// TIA Portal project "Diarator_V2" (V16)

(* hardware
DEVICE "S7-1200 station_1"  S7-1200 Station
   slot 0: "Rack_0"  S7-1200 Rack  Rack  V1.0
   slot 1: "PLC_1"  CPU 1214C DC/DC/Rly  6ES7 214-1HG40-0XB0  V4.4
   slot 2: "DI 16/DQ 16x24VDC_2"  SM 1223 DI8/DQ8 x relay  6ES7 223-1PH32-0XB0  V2.0
   slot 3: "AI 4x13BIT_1"  6ES7 231-4HD32-0XB0  V2.1
   slot 4: "AI 4x13BIT_2"  6ES7 231-4HD32-0XB0  V2.1
   slot 5: "AQ 4x14BIT_1"  6ES7 232-4HD32-0XB0  V2.1
*)

// ===== PLC "PLC_1"  CPU 1214C DC/DC/Rly =====

VAR_GLOBAL   // PLC tag table "Default tag table"
   "rAlarm_SetMinPressSteam" AT %MW12 : Int;   // Уставка минимального давления пара
   "rAI_Press1" AT %MW14 : Int;   // Давление датчика
   "bAlarmPress1" AT %M16.0 : Bool;
   "rAlarm_SetMinPressWater" AT %MW18 : Int;   // Уставка аварийного давления воды
   "rAI_Press2" AT %MW20 : Int;
   "1_MTrig" AT %M6.4 : Bool;
   "2_MTrig" AT %M6.5 : Bool;
   "3_MTrig" AT %M6.6 : Bool;
   "mTrig1" AT %M7.0 : Bool;
   "mTrig" AT %M1.4 : Bool;
END_VAR

VAR_GLOBAL   // PLC tag table "HMI_"
   "bHMI_button_Start" AT %M2.0 : Bool;   // Кнопка старт
   "bHMI_button_Stop" AT %M2.1 : Bool;   // Кнопка стоп
   "bHMI_button_Pause" AT %M2.2 : Bool;   // Кнопка пауза
   "bStartAllowed" AT %M100.0 : Bool;   // Готовность к старту
   "bOpenWindStartConveyor" AT %M100.1 : Bool;   // Вызов окна подтверждения оператором старта конвейера
   "iHMI_Num_StatrPaster" AT %MW4 : Int;
   "bTypePID_Zone1" AT %M8.0 : Bool;   // Тип ПИД - 1 - Охлаждение, 0 - Нагрев
   "bTypePID_Zone2" AT %M8.1 : Bool;   // Тип ПИД - 1 - Охлаждение, 0 - Нагрев
   "bTypePID_Zone3" AT %M8.2 : Bool;   // Тип ПИД - 1 - Охлаждение, 0 - Нагрев
   "bTypePID_Zone4" AT %M8.3 : Bool;   // Тип ПИД - 1 - Охлаждение, 0 - Нагрев
   "bTypePID_Zone5" AT %M8.4 : Bool;   // Тип ПИД - 1 - Охлаждение, 0 - Нагрев
   "bAllAuto" AT %M0.6 : Bool;   // Перевод всего оборудования в авто с ручного
   "bZoomerOff" AT %M0.7 : Bool;   // Выкл пищалка
   "bResetAlarmCommon" AT %M6.0 : Bool;   // Общий сброс аварий
   "bResCountWaterO2" AT %M0.5 : Bool;   // Сброс счетчика готовой воды
   "bCountWaterToSewerge" AT %MW72 : Int;   // Счетчики воды в канализацию
   "bCountWaterToReadyO2" AT %MD10 : DInt;   // Счетчикиготовой водыО2
   "bHMI_ResetCounterAll_Water" AT %M3.2 : Bool;   // Кнопка сброса счетчика воды общего
   "iCount_All_Water" AT %MD62 : UDInt;   // Значение общего кол-ва воды пройденного через счетчик
   "iCount_CIP_AlL" AT %MD126 : UDInt;   // Счетчик СИП
   "bResCount_CIP" AT %M3.3 : Bool;   // Кнопка Сброса счетчика СИП
   "iStatusWork" AT %MW76 : Int;   // 0 - стоп 1 - СИП 2 - ДИаратор Подготовка 4 - Диаратор производство Статус работы для панели
   "timeStart" AT %MD50 : DInt;   // Задержка стоп/старт насосы
   "timeAlarmNoWater" AT %MD54 : DInt;   // Авария при длительной отстутвии воды
   "bDryContrlPump_1" AT %M78.0 : Bool;   // Контроль сухого хода насоса 1
   "bResTimeWorkSystem" AT %M6.7 : Bool;   // Сброс времени наработки системой
   "iOurs_WorkSystem" AT %MW120 : UInt;   // Часы работы системы
   "iMini_WorkSystem" AT %MW122 : Int;   // Мин работы системы
   "iSec_WorkSystem" AT %MW124 : Int;   // Секунды работы системы
END_VAR

VAR_GLOBAL   // PLC tag table "DI"
   "DI_0.0_Кнопка экстренной остановки E-Stop №1" AT %I0.0 : Bool;
   "DI_0.1_Положение ВОДА" AT %I0.1 : Bool;
   "DI_0.2_Положение СИП" AT %I0.2 : Bool;
   "DI_0.3_Клапан V1" AT %I0.3 : Bool;
   "DI_0.4_Клапан V3" AT %I0.4 : Bool;   // Импльс от расходомера
   "DI_0.5_Клапан V4" AT %I0.5 : Bool;
   "DI_0.6_Клапан V5" AT %I0.6 : Bool;
   "DI_0.7_Клапан V6" AT %I0.7 : Bool;
   "DI_1.0_LS1" AT %I1.0 : Bool;
   "DI_1.1_LS2" AT %I1.1 : Bool;
   "DI_1.2_LS3" AT %I1.2 : Bool;
   "DI_1.3_LS4" AT %I1.3 : Bool;
   "DI_1.4_Реле давления воздуха" AT %I1.4 : Bool;
   "DI_1.5_Импульсы Расходомера" AT %I1.5 : Bool;
   "DI_2.0_Автомат_1" AT %I2.0 : Bool;
   "DI_2.1_Работа_Частотник_1" AT %I2.1 : Bool;
   "DI_2.2_Автомат_2" AT %I2.2 : Bool;
   "DI_2.3_Работа_Частотник_2" AT %I2.3 : Bool;
END_VAR

VAR_GLOBAL   // PLC tag table "MyTags"
   "Разрешение работы конвейера" AT %M0.0 : Bool;   // Команда разрешения от Глобального блока работы
   "bMain_AlarmSystem" AT %M2.3 : Bool;   // АВария в системе (Общая)
   "bStartWork_Main" AT %M1.7 : Bool;   // Старт Общий Диаэратор
   "bPosition_Diarator" AT %M3.0 : Bool;   // Калачи в положении Диаэратор
   "bPosition_CIP" AT %M3.1 : Bool;   // Калачи в положении СИП
   "bReady_O2" AT %M1.3 : Bool;   // Готовность воды по датчику кислорода
   "bDiarator_WaterReady" AT %M0.2 : Bool;   // Меркер готовности диаратора по счетчику
   "bTypeControlO2" AT %M1.2 : Bool;   // Переключение типа контроля О2 (счетик - 0, датчик О2 - 1)
   "bImpulseFlow" AT %M3.4 : Bool;   // Импульс расходомера
   "diAccumTime" AT %MD116 : DInt;   // Аккумулятор времени работы установки
   "TestReset" AT %M7.1 : Bool;   // Блок аварий для тестов
   "bPaus" AT %M1.1 : Bool;
   "MTrig2" AT %M7.2 : Bool;
   "TestDI" AT %M0.4 : Bool;
   "m_STOP" AT %M1.6 : Bool;
   "_bCloseFV_CIP" AT %M1.0 : Bool;
END_VAR

VAR_GLOBAL   // PLC tag table "Timers_CPU"
   "Time_0.1s" AT %M500.0 : Bool;
   "Time_0.2s" AT %M500.1 : Bool;
   "Time_0.4s" AT %M500.2 : Bool;
   "Time_0.5s" AT %M500.3 : Bool;
   "Time_0.8s" AT %M500.4 : Bool;
   "Time_1s" AT %M500.5 : Bool;
   "Time_1.6s" AT %M500.6 : Bool;
   "Time_2s" AT %M500.7 : Bool;
END_VAR

VAR_GLOBAL   // PLC tag table "DO"
   "DO_0.0_Пневмо_остров клапан 1" AT %Q0.0 : Bool;
   "DO_0.1_Пневмо_остров клапан 2" AT %Q0.1 : Bool;
   "DO_0.2_Пневмо_остров клапан 3" AT %Q0.2 : Bool;
   "DO_0.3_Пневмо_остров клапан 4" AT %Q0.3 : Bool;
   "DO_0.4_Пневмо_остров клапан 5" AT %Q0.4 : Bool;
   "DO_0.5_Пневмо_остров клапан 6" AT %Q0.5 : Bool;
   "DO_0.6_Пневмо_остров клапан 7" AT %Q0.6 : Bool;
   "DO_0.7_Пневмо_остров клапан 8" AT %Q0.7 : Bool;
   "DO_0.8_Пневмо_остров клапан 9" AT %Q1.0 : Bool;
   "DO_0.9_Пневмо_остров клапан 10" AT %Q1.1 : Bool;
   "Преобразователь частоты 1 пуск" AT %Q2.4 : Bool;
   "Преобразователь частоты 2 пуск" AT %Q2.5 : Bool;
   "Световая колонна - зеленый" AT %Q2.0 : Bool;
   "Световая колонна - желтый" AT %Q2.1 : Bool;
   "Световая колонна - красный" AT %Q2.2 : Bool;
   "Выход_Готовность ВОДА" AT %Q2.6 : Bool;
   "Выход_Готовность СИП" AT %Q2.7 : Bool;
END_VAR

VAR_GLOBAL   // PLC tag table "AI"
   "ТТ01" AT %IW120 : Int;   // Температура
   "FIC" AT %IW112 : Int;   // Расходомер
   "PT-01" AT %IW114 : Int;   // Давление 1
   "PT-02" AT %IW116 : Int;   // Давление 2
   "PT-03" AT %IW118 : Int;   // Давление 3
   "O2" AT %IW124 : Int;   // Датчик Кислорода О2
   "ТТ02_FromO2" AT %IW126 : Int;   // Температура
END_VAR

VAR_GLOBAL   // PLC tag table "AO"
   "AO_0.0_Преобразователь частоты 1" AT %QW144 : Int;
   "AO_0.1_Преобразователь частоты 2" AT %QW146 : Int;
   "AO_0.2_Управляемый клапан №2" AT %QW148 : Int;
END_VAR

VAR_GLOBAL   // PLC tag table "_TEst_1"
   "test_stateDiar" AT %M0.1 : Bool;
   "test_PressSensor" AT %MD22 : Real;
END_VAR

TYPE "FV_o/c"
   STRUCT
      bOpenCmd : Bool;   // Команда открыть (автомат)
      bManualMode : Bool;   // Ручной режим (TRUE)
      bManualOpen : Bool;   // Команда открыть в ручном режиме
      bFeedbackOpen : Bool;   // Обратная связь "Открыт"
      tMaxTime : DInt;   // Время на открытие
      bResetAlarm : Bool;   // Сброс аварии
      bCheckFeedback : Bool;   // Выбирается есть ли обратная связь у клапана
      bOutOpen : Bool;   // Выход на открытие клапана
      iOutState : Int;   // Выход статуса клапана
   END_STRUCT;
END_TYPE

TYPE "PID_Param"
   STRUCT
      bModeActivate : Bool;   // Запуск выбранного типа работы
      iModeNum : Int := 3;   // 0 -стоп 1 - автонастройка 2 -точная автонастройка 3 - авто режим 4 - ручной режим
      iOutState : Int;   // В каком режиме ПИД
      bOutError : Bool;   // Выход при ошибке TRUE
      iOutErrorBits : Int;   // Бит с кодом ошибки (см. мануал)
      iProgress : Int;   // Состояние в % при автонастройки, сколько сделано
   END_STRUCT;
END_TYPE

TYPE "FV_regul"
   STRUCT
      bHMI_ManualMode : Bool;   // Переключение режима авто/ручно (0 - А, 1 - Р)
      rHMI_ManualSet : Real;   // Уставка в ручном режиме (0-100)
      rAuto_Set : Real;   // Уставка в автоматическом режиме
      iOut_AO : Int;   // Сигнал на аналоговый выход
      "rHMI_Out_FV-%" : Real;   // Состояние в % (0-100)
      bOut_DO_ValveOpen : Bool;   // Дискретный сигнал открытия
   END_STRUCT;
END_TYPE

TYPE "Коэф ПИД"
   STRUCT
      Gain : Int;   // Коэф П
      I : DInt;   // Коэф И
      D : DInt;   // Коэф Д
   END_STRUCT;
END_TYPE

TYPE "tipe_Pumps"
   STRUCT
      bAutoStartPump : Bool;   // Старт в автоматическом режиме
      rAutoSpeedPump : Real;   // Скорость в автоматическом режиме
      bManualMode : Bool;   // Ручной режим вкл/выкл
      bManualStart : Bool;   // Старт в ручном режиме
      rManualSpeed : Real;   // Скорость в ручном режиме
      rHMI_Speed : Real;   // Выходная скороость для HMI
      bHMI_PumpRun : Bool;   // Статус работы для HMI
      bresAlarm : Bool;   // Сброс аварий
      iStatusPump : Int;   // Статус насоса
   END_STRUCT;
END_TYPE

TYPE "Tipe_DI"
   STRUCT
      f_DI_out : Bool;
      "bFiltr_on/off" : Bool := true;
      diTime_filtr : Time := T#100ms;
      bSimulation : Bool;   // Включение режима симуляции
      "bSim_On/Off" : Bool;   // Управление симуляцией
   END_STRUCT;
END_TYPE

TYPE "Tipe_AI"
   STRUCT
      bSimulate : Bool;   // Вкл симуляции датчика
      rSimulateValue : Real;   // Значение симуляции датчика
      rSensor_HL : Real;   // Верхний предел датчика
      rSensor_LL : Real;   // Нижний предел датчика
      bFiltr : Bool;   // Управление фильтром значений
      rAI_Value : Real;   // Значение аналогового датчика
   END_STRUCT;
END_TYPE

// folder: AI_Signal/AI_DB/4-20

DATA_BLOCK "AI_(4-20)_1_DB_1"   // DB16
{ S7_Optimized_Access := 'FALSE' }
VERSION : 0.1
// stored: InstanceOfName AI_(4-20)_1
"AI_(4-20)_1"
BEGIN
   HMI_rParam_Sensor_HL := 100.0;
   HMI_rParam_Sensor_LL := -50.0;
END_DATA_BLOCK

DATA_BLOCK "AI_(4-20)_1_DB_2"   // DB17
{ S7_Optimized_Access := 'FALSE' }
VERSION : 0.1
// stored: InstanceOfName AI_(4-20)_1
"AI_(4-20)_1"
BEGIN
END_DATA_BLOCK

DATA_BLOCK "AI_(4-20)_1_DB_4"   // DB18
{ S7_Optimized_Access := 'FALSE' }
VERSION : 0.1
// stored: InstanceOfName AI_(4-20)_1
"AI_(4-20)_1"
BEGIN
   HMI_rParam_Sensor_HL := 6.0;
END_DATA_BLOCK

DATA_BLOCK "AI_(4-20)_1_DB_3"   // DB27
{ S7_Optimized_Access := 'FALSE' }
VERSION : 0.1
// stored: InstanceOfName AI_(4-20)_1
"AI_(4-20)_1"
BEGIN
   HMI_rParam_Sensor_HL := 100.0;
END_DATA_BLOCK

DATA_BLOCK "AI_(4-20)_1_DB_5"   // DB28
{ S7_Optimized_Access := 'FALSE' }
VERSION : 0.1
// stored: InstanceOfName AI_(4-20)_1
"AI_(4-20)_1"
BEGIN
   HMI_rParam_Sensor_HL := 6.0;
END_DATA_BLOCK

DATA_BLOCK "AI_(4-20)_1_DB_6"   // DB60
{ S7_Optimized_Access := 'FALSE' }
VERSION : 0.1
// stored: InstanceOfName AI_(4-20)_1
"AI_(4-20)_1"
BEGIN
END_DATA_BLOCK

DATA_BLOCK "AI_(4-20)_1_DB_7"   // DB61
{ S7_Optimized_Access := 'FALSE' }
VERSION : 0.1
// stored: InstanceOfName AI_(4-20)_1
"AI_(4-20)_1"
BEGIN
END_DATA_BLOCK

// folder: DB-FB

DATA_BLOCK "FB_check_For_Start_DB"   // DB1
{ S7_Optimized_Access := 'FALSE' }
VERSION : 0.1
// stored: InstanceOfName FB_check_For_Start
"FB_check_For_Start"
BEGIN
END_DATA_BLOCK

DATA_BLOCK "FB_Emergency_DB"   // DB3
{ S7_Optimized_Access := 'FALSE' }
VERSION : 0.1
// stored: InstanceOfName FB_Аварии
"FB_Аварии"
BEGIN
END_DATA_BLOCK

DATA_BLOCK "Tank_Diarator_DB"   // DB11
{ S7_Optimized_Access := 'TRUE' }
VERSION : 0.1
// stored: InstanceOfName Tank_Diarator
"Tank_Diarator"
BEGIN
END_DATA_BLOCK

DATA_BLOCK "FB_Control_O2_DB"   // DB12
{ S7_Optimized_Access := 'TRUE' }
VERSION : 0.1
// stored: InstanceOfName FB_Control_O2
"FB_Control_O2"
BEGIN
END_DATA_BLOCK

DATA_BLOCK "FB_Tank_2(Buffer)_DB"   // DB13
{ S7_Optimized_Access := 'TRUE' }
VERSION : 0.1
// stored: InstanceOfName FB_Tank_2(Buffer)
"FB_Tank_2(Buffer)"
BEGIN
END_DATA_BLOCK

DATA_BLOCK "FB_Control_Press_Tank2_DB"   // DB14
{ S7_Optimized_Access := 'TRUE' }
VERSION : 0.1
// stored: InstanceOfName FB_Control_Press_Tank2
"FB_Control_Press_Tank2"
BEGIN
END_DATA_BLOCK

DATA_BLOCK "FB_CIP_DB"   // DB15
{ S7_Optimized_Access := 'TRUE' }
VERSION : 0.1
// stored: InstanceOfName FB_CIP
"FB_CIP"
BEGIN
END_DATA_BLOCK

DATA_BLOCK "FB_OwerPress_Tank_2_DB"   // DB64
{ S7_Optimized_Access := 'FALSE' }
VERSION : 0.1
// stored: InstanceOfName FB_OwerPress_Tank_2
"FB_OwerPress_Tank_2"
BEGIN
END_DATA_BLOCK

DATA_BLOCK "FB_SVETOFOR_DB"   // DB102
{ S7_Optimized_Access := 'TRUE' }
VERSION : 0.1
// stored: InstanceOfName FB_SVETOFOR
"FB_SVETOFOR"
BEGIN
END_DATA_BLOCK

// folder: DI_signal/DB_DI

DATA_BLOCK "LS-1"   // DB33
{ S7_Optimized_Access := 'FALSE' }
VERSION : 0.1
// stored: InstanceOfName FB_DI_Pointer
"FB_DI_Pointer"
BEGIN
END_DATA_BLOCK

DATA_BLOCK "LS-2"   // DB35
{ S7_Optimized_Access := 'FALSE' }
VERSION : 0.1
// stored: InstanceOfName FB_DI_Pointer
"FB_DI_Pointer"
BEGIN
END_DATA_BLOCK

DATA_BLOCK "LS-3"   // DB36
{ S7_Optimized_Access := 'FALSE' }
VERSION : 0.1
// stored: InstanceOfName FB_DI_Pointer
"FB_DI_Pointer"
BEGIN
END_DATA_BLOCK

DATA_BLOCK "LS-4"   // DB46
{ S7_Optimized_Access := 'FALSE' }
VERSION : 0.1
// stored: InstanceOfName FB_DI_Pointer
"FB_DI_Pointer"
BEGIN
END_DATA_BLOCK

DATA_BLOCK "P1_ControlWorking"   // DB47
{ S7_Optimized_Access := 'FALSE' }
VERSION : 0.1
// stored: InstanceOfName FB_DI_Pointer
"FB_DI_Pointer"
BEGIN
END_DATA_BLOCK

DATA_BLOCK "DI_EStop1"   // DB48
{ S7_Optimized_Access := 'FALSE' }
VERSION : 0.1
// stored: InstanceOfName FB_DI
"FB_DI"
BEGIN
END_DATA_BLOCK

DATA_BLOCK "State_Water"   // DB49
{ S7_Optimized_Access := 'FALSE' }
VERSION : 0.1
// stored: InstanceOfName FB_DI
"FB_DI"
BEGIN
END_DATA_BLOCK

DATA_BLOCK "State_CIP"   // DB50
{ S7_Optimized_Access := 'FALSE' }
VERSION : 0.1
// stored: InstanceOfName FB_DI
"FB_DI"
BEGIN
END_DATA_BLOCK

DATA_BLOCK "FeedBack_V1"   // DB51
{ S7_Optimized_Access := 'FALSE' }
VERSION : 0.1
// stored: InstanceOfName FB_DI
"FB_DI"
BEGIN
END_DATA_BLOCK

DATA_BLOCK "Feedback_V3"   // DB52
{ S7_Optimized_Access := 'FALSE' }
VERSION : 0.1
// stored: InstanceOfName FB_DI
"FB_DI"
BEGIN
END_DATA_BLOCK

DATA_BLOCK "Feedback_V4"   // DB53
{ S7_Optimized_Access := 'FALSE' }
VERSION : 0.1
// stored: InstanceOfName FB_DI
"FB_DI"
BEGIN
END_DATA_BLOCK

DATA_BLOCK "FeedBack_V5"   // DB54
{ S7_Optimized_Access := 'FALSE' }
VERSION : 0.1
// stored: InstanceOfName FB_DI
"FB_DI"
BEGIN
END_DATA_BLOCK

DATA_BLOCK "FeedBack_V6"   // DB55
{ S7_Optimized_Access := 'FALSE' }
VERSION : 0.1
// stored: InstanceOfName FB_DI
"FB_DI"
BEGIN
END_DATA_BLOCK

DATA_BLOCK "PressAir"   // DB78
{ S7_Optimized_Access := 'FALSE' }
VERSION : 0.1
// stored: InstanceOfName FB_DI_Pointer
"FB_DI_Pointer"
BEGIN
END_DATA_BLOCK

DATA_BLOCK "ImpFlow"   // DB79
{ S7_Optimized_Access := 'FALSE' }
VERSION : 0.1
// stored: InstanceOfName FB_DI_Pointer
"FB_DI_Pointer"
BEGIN
END_DATA_BLOCK

DATA_BLOCK "CircuitControl-1"   // DB80
{ S7_Optimized_Access := 'FALSE' }
VERSION : 0.1
// stored: InstanceOfName FB_DI_Pointer
"FB_DI_Pointer"
BEGIN
END_DATA_BLOCK

DATA_BLOCK "CircuitControl-2"   // DB81
{ S7_Optimized_Access := 'FALSE' }
VERSION : 0.1
// stored: InstanceOfName FB_DI_Pointer
"FB_DI_Pointer"
BEGIN
END_DATA_BLOCK

DATA_BLOCK "P2_ControlWorking"   // DB82
{ S7_Optimized_Access := 'FALSE' }
VERSION : 0.1
// stored: InstanceOfName FB_DI_Pointer
"FB_DI_Pointer"
BEGIN
END_DATA_BLOCK

// folder: FB/R_TRIG_DB

DATA_BLOCK "R_trig_All_Auto"   // DB40
{ S7_Optimized_Access := 'TRUE' }
VERSION : 0.1
// stored: InstanceOfName R_trig
"R_trig"
BEGIN
END_DATA_BLOCK

DATA_BLOCK "R_trig_DB_Stop_CIP"   // DB56
{ S7_Optimized_Access := 'TRUE' }
VERSION : 0.1
// stored: InstanceOfName R_trig
"R_trig"
BEGIN
END_DATA_BLOCK

DATA_BLOCK "R_trig_ResTimeWorkSystem"   // DB58
{ S7_Optimized_Access := 'TRUE' }
VERSION : 0.1
// stored: InstanceOfName R_trig
"R_trig"
BEGIN
END_DATA_BLOCK

DATA_BLOCK "R_trig_DB"   // DB99
{ S7_Optimized_Access := 'TRUE' }
VERSION : 0.1
// stored: InstanceOfName R_trig
"R_trig"
BEGIN
END_DATA_BLOCK

DATA_BLOCK "R_trig_DB_Alarm_Zoomer"   // DB101
{ S7_Optimized_Access := 'TRUE' }
VERSION : 0.1
// stored: InstanceOfName R_trig
"R_trig"
BEGIN
END_DATA_BLOCK

DATA_BLOCK "R_trig_DB_Pause"   // DB103
{ S7_Optimized_Access := 'TRUE' }
VERSION : 0.1
// stored: InstanceOfName R_trig
"R_trig"
BEGIN
END_DATA_BLOCK

// folder: System blocks/Program resources

DATA_BLOCK "IEC_Counter_ReadyWaterO2"   // DB29
{ S7_Optimized_Access := 'TRUE' }
AUTHOR : SIMATIC
FAMILY : IEC
NAME : DCNTR
VERSION : 1.2
// stored: InstanceOfName IEC_DCOUNTER
"IEC_DCOUNTER"
BEGIN
END_DATA_BLOCK

DATA_BLOCK "IEC_Counter_DiarSewerage"   // DB31
{ S7_Optimized_Access := 'TRUE' }
AUTHOR : Simatic
FAMILY : IEC
NAME : CNTR
VERSION : 1.0
// stored: InstanceOfName IEC_COUNTER
"IEC_COUNTER"
BEGIN
END_DATA_BLOCK

DATA_BLOCK "IEC_Counter_All_Water"   // DB37
{ S7_Optimized_Access := 'TRUE' }
AUTHOR : Simatic
FAMILY : IEC
NAME : UDCNTR
VERSION : 1.2
// stored: InstanceOfName IEC_UDCOUNTER
"IEC_UDCOUNTER"
BEGIN
END_DATA_BLOCK

DATA_BLOCK "IEC_Counter_CIP"   // DB38
{ S7_Optimized_Access := 'TRUE' }
AUTHOR : Simatic
FAMILY : IEC
NAME : UCNTR
VERSION : 1.2
// stored: InstanceOfName IEC_UCOUNTER
"IEC_UCOUNTER"
BEGIN
END_DATA_BLOCK

DATA_BLOCK "IEC_Timer_DetectDry_1"   // DB42
{ S7_Optimized_Access := 'TRUE' }
AUTHOR : Simatic
FAMILY : IEC
NAME : IEC_TMR
VERSION : 1.0
// stored: InstanceOfName IEC_TIMER
"IEC_TIMER"
BEGIN
END_DATA_BLOCK

DATA_BLOCK "IEC_Timer_ResDrySens"   // DB45
{ S7_Optimized_Access := 'TRUE' }
AUTHOR : Simatic
FAMILY : IEC
NAME : IEC_TMR
VERSION : 1.0
// stored: InstanceOfName IEC_TIMER
"IEC_TIMER"
BEGIN
END_DATA_BLOCK

DATA_BLOCK "IEC_Counter_0_DB"   // DB59
{ S7_Optimized_Access := 'TRUE' }
AUTHOR : Simatic
FAMILY : IEC
NAME : CNTR
VERSION : 1.0
// stored: InstanceOfName IEC_COUNTER
"IEC_COUNTER"
BEGIN
END_DATA_BLOCK

DATA_BLOCK "IEC_Timer_0_DB"   // DB62
{ S7_Optimized_Access := 'TRUE' }
AUTHOR : Simatic
FAMILY : IEC
NAME : IEC_TMR
VERSION : 1.0
// stored: InstanceOfName IEC_TIMER
"IEC_TIMER"
BEGIN
END_DATA_BLOCK

// folder: Use VARs to HMI

DATA_BLOCK "DB2_HMI_SET"   // DB2
{ S7_Optimized_Access := 'FALSE' }
VERSION : 0.1
   VAR
      rO2_SP : Real;   // Уставка для датчика кислорода
      rHisteresis_O2_SP : Real;   // Уставка гистерезиса для допустим отклонения О2
      diTimeLost_Gist_O2 : DInt;   // Уставка времени ожидания при выходе за пределы уставки
      rFlow_SP : Int;   // Уставка расхода воды готовности по счетчику
      diTimeToReadyO2 : DInt;   // Уставка ожидания перехода в готовность воды при достижении уставки О2
      rPT02_SP : Real;   // Уставка давления в танке 2
      rPT02_OwerPress_SP : Real;   // Уставка слишком высокого давления Танк 2
      rPT02_Hister_OwerPress : Real;   // Уставка гистерезиса
      diTimeToOpenValveCO2 : DInt := 2;   // Время отсчета для открытия клапана при понижении давления в Такнке 2
      diTimeToCloseValveCO2 : DInt := 2;   // Время отсчета для закрытия клапана при возвращении давления в Такнке 2
      diFlipTimeCIP : DInt := 3;   // Время задержки между переходом флипования
      diFlipPauseFlipeCIP : DInt := 2;   // Время задержки перед началом цикла флипования
      rSetValve_2_OUT : Real;   // Уставка расхода для клапана 2 задание для клапана
      rSetValve_2_Diarator : Real := 3000.0;   // Уставка клапана 2 при режиме ДИаратор
      rSetValve_2_CIP : Real := 5000.0;   // Уставка клапана 2 при режиме СИП
      "rSetPump-1_OUT" : Real;   // Уставка для насоса 1 - OUT
      "rSetPump-1_Diarator" : Real := 30.0;   // Уставка для насоса 1 - Диаратор
      "rSetPump-1_CIP" : Real := 20.0;   // Уставка для насоса 1 - CIP
      "rSetPump-2_OUT" : Real;   // Уставка для насоса 2 - OUT
      "rSetPump-2_Diarator" : Real := 3.0;   // Уставка для насоса 2 - Диаратор
      "rSetPump-2_CIP" : Real := 3.0;   // Уставка для насоса 2 - CIP
      rDetectDry_PressTank1_SP : Real := 2.0;   // Уставка обнаружения сухого хода для насоса 1
      diTimeDetectDrt : DInt := 2;   // Время для обнаружения сухого хода
      Di_timeCloseFV : DInt := 5000;   // Время задержки закрытия клапанов в режиме СИП при "СТОП"
      rLewelTank1_Stop : Real;   // Уровень емкости - закрытие Кл1
      rLewelTank1_Start : Real;   // Уровень емкости - открытие Кл1
   END_VAR
BEGIN
END_DATA_BLOCK

DATA_BLOCK "FVs_o/p"   // DB6
{ S7_Optimized_Access := 'FALSE' }
VERSION : 0.1
   VAR
      FV_1 : "FV_o/c";
      FV_2 : "FV_o/c";
      FV_3 : "FV_o/c";
      FV_4 : "FV_o/c";
      FV_5 : "FV_o/c";
      FV_6 : "FV_o/c";
      FV_7 : "FV_o/c";
      FV_8 : "FV_o/c";
      FV_9 : "FV_o/c";
      FV_10 : "FV_o/c";
   END_VAR
BEGIN
END_DATA_BLOCK

DATA_BLOCK "FVs_Regul"   // DB24
{ S7_Optimized_Access := 'FALSE' }
VERSION : 0.1
   VAR
      FV_Regul_1 : "FV_regul";
   END_VAR
BEGIN
END_DATA_BLOCK

DATA_BLOCK "Pumps"   // DB30
{ S7_Optimized_Access := 'FALSE' }
VERSION : 0.1
   VAR
      Pump_1 : "tipe_Pumps";
      Pump_2 : "tipe_Pumps";
   END_VAR
BEGIN
END_DATA_BLOCK

DATA_BLOCK "LS"   // DB34
{ S7_Optimized_Access := 'FALSE' }
VERSION : 0.1
   VAR
      "LS-1" : Bool;   // Уровень емкости 1 колонны
      "LS-2" : Bool;   // Нижний уровень 2 колонны
      "LS-3" : Bool;   // Средний уровень 2 колонны
      "LS-4" : Bool;   // Верхний уровень 2 колонны
   END_VAR
BEGIN
END_DATA_BLOCK

DATA_BLOCK "DI"   // DB43
{ S7_Optimized_Access := 'FALSE' }
VERSION : 0.1
   VAR
      DI_0 : "Tipe_DI";   // Stop_Button
      DI_1 : "Tipe_DI";   // Water_State
      DI_2 : "Tipe_DI";   // CIP_State
      DI_3 : "Tipe_DI";   // Feedback_V1
      DI_4 : "Tipe_DI";   // Feedback_V3
      DI_5 : "Tipe_DI";   // Feedback_V4
      DI_6 : "Tipe_DI";   // Feedback_V5
      DI_7 : "Tipe_DI";   // Feedback_V6
      DI_8 : "Tipe_DI";   // LS-1
      DI_9 : "Tipe_DI";   // LS-2
      DI_10 : "Tipe_DI";   // LS-3
      DI_11 : "Tipe_DI";   // LS-4
      DI_12 : "Tipe_DI";   // PressAir_Rele
      DI_13 : "Tipe_DI";   // Impuls_CounterFlow
      DI_14 : "Tipe_DI";   // Доп контакт автомата 1
      DI_15 : "Tipe_DI";   // StatusWorkPump1
      DI_16 : "Tipe_DI";   // Доп контакт автомата 2
      DI_17 : "Tipe_DI";   // StatusWorkPump2
      DI_18 : "Tipe_DI";
      DI_19 : "Tipe_DI";
      DI_20 : "Tipe_DI";
      DI_21 : "Tipe_DI";
      DI_22 : "Tipe_DI";
      DI_23 : "Tipe_DI";
      DI_24 : "Tipe_DI";
      DI_25 : "Tipe_DI";
      DI_26 : "Tipe_DI";
      DI_27 : "Tipe_DI";
      DI_28 : "Tipe_DI";
      DI_29 : "Tipe_DI";
      DI_30 : "Tipe_DI";
   END_VAR
BEGIN
END_DATA_BLOCK

DATA_BLOCK "PID_State_Param"   // DB57
{ S7_Optimized_Access := 'FALSE' }
VERSION : 0.1
   VAR
      PID_Vavle2 : "PID_Param";
      PID_Pump1 : "PID_Param";
      PID_Pump2 : "PID_Param";
   END_VAR
BEGIN
END_DATA_BLOCK

DATA_BLOCK "Alarms"   // DB87
{ S7_Optimized_Access := 'FALSE' }
VERSION : 0.1
   VAR
      Ai_Alarm : Array[1..8] of Struct   // Аварии датчиков аналоговых
         ALARM : Bool;
         RESET : Bool;
      END_STRUCT;
      Pump_Alarm : Array[1..5] of Struct   // Аварии насосов
         ALARM : Bool;
         RESET : Bool;
      END_STRUCT;
      Avtomat_Off : Array[1..2] of Struct   // Контроль состояния вкл мотор автоматов
         ALARM : Bool;
      END_STRUCT;
      FV_Alarm : Array[1..10] of Struct   // Авария клапанов
         ALARM : Bool;
         RESET : Bool;
      END_STRUCT;
      "xE-Stop_1" : Bool;   // Авария по кнопке 1
      xVoltRele : Bool;   // Авария реле контроля фаз
      xLongWaitWater : Bool;   // Авария, долгое ожидание заполнения нижнего уровня емкости
      xPressAir : Bool;   // Авария реле давления воздуха
   END_VAR
BEGIN
END_DATA_BLOCK

DATA_BLOCK "AI_DB"   // DB90
{ S7_Optimized_Access := 'FALSE' }
VERSION : 0.1
   VAR
      TT_01 : "Tipe_AI";   // Температура
      FIC : "Tipe_AI";   // Расходомер
      PT_01 : "Tipe_AI";   // Давление Емкость_1
      PT_02 : "Tipe_AI";   // Давление Емкость_2
      PT_03 : "Tipe_AI";   // Давление Выход с емкости
      ТТ02_FromO2 : "Tipe_AI";   // Значение температуры с датчика кислорода
      O2 : "Tipe_AI";   // Кислород
   END_VAR
BEGIN
   O2.rSensor_HL := 10.0;
   O2.bFiltr := true;
   TT_01.bFiltr := true;
   FIC.bFiltr := true;
   PT_01.bFiltr := true;
   PT_02.bFiltr := true;
   PT_03.bFiltr := true;
   TT_01.rSensor_HL := 100.0;
   TT_01.rSensor_LL := -50.0;
   PT_01.rSensor_HL := 1.0;
   PT_02.rSensor_HL := 6.0;
   PT_03.rSensor_HL := 6.0;
END_DATA_BLOCK

// folder: Клапана/FV_o/C/FV_DB

DATA_BLOCK "FV_1"   // DB4
{ S7_Optimized_Access := 'FALSE' }
VERSION : 0.1
// stored: InstanceOfName Valve(c/o)
"Valve(c/o)"
BEGIN
END_DATA_BLOCK

DATA_BLOCK "FV_5"   // DB5
{ S7_Optimized_Access := 'FALSE' }
VERSION : 0.1
// stored: InstanceOfName Valve(c/o)
"Valve(c/o)"
BEGIN
END_DATA_BLOCK

DATA_BLOCK "FV_6"   // DB7
{ S7_Optimized_Access := 'FALSE' }
VERSION : 0.1
// stored: InstanceOfName Valve(c/o)
"Valve(c/o)"
BEGIN
END_DATA_BLOCK

DATA_BLOCK "FV_7"   // DB8
{ S7_Optimized_Access := 'FALSE' }
VERSION : 0.1
// stored: InstanceOfName Valve(c/o)
"Valve(c/o)"
BEGIN
END_DATA_BLOCK

DATA_BLOCK "FV_2"   // DB9
{ S7_Optimized_Access := 'FALSE' }
VERSION : 0.1
// stored: InstanceOfName Valve(c/o)
"Valve(c/o)"
BEGIN
END_DATA_BLOCK

DATA_BLOCK "FV_3"   // DB10
{ S7_Optimized_Access := 'FALSE' }
VERSION : 0.1
// stored: InstanceOfName Valve(c/o)
"Valve(c/o)"
BEGIN
END_DATA_BLOCK

DATA_BLOCK "FV_4"   // DB19
{ S7_Optimized_Access := 'FALSE' }
VERSION : 0.1
// stored: InstanceOfName Valve(c/o)
"Valve(c/o)"
BEGIN
END_DATA_BLOCK

DATA_BLOCK "FV_8"   // DB21
{ S7_Optimized_Access := 'FALSE' }
VERSION : 0.1
// stored: InstanceOfName Valve(c/o)
"Valve(c/o)"
BEGIN
END_DATA_BLOCK

DATA_BLOCK "FV_9"   // DB22
{ S7_Optimized_Access := 'FALSE' }
VERSION : 0.1
// stored: InstanceOfName Valve(c/o)
"Valve(c/o)"
BEGIN
END_DATA_BLOCK

DATA_BLOCK "FV_10"   // DB23
{ S7_Optimized_Access := 'FALSE' }
VERSION : 0.1
// stored: InstanceOfName Valve(c/o)
"Valve(c/o)"
BEGIN
END_DATA_BLOCK

// folder: Клапана/FV_regul/DB

DATA_BLOCK "FV_Regul_1_DB"   // DB20
{ S7_Optimized_Access := 'FALSE' }
VERSION : 0.1
// stored: InstanceOfName Valve(regul)
"Valve(regul)"
BEGIN
END_DATA_BLOCK

// folder: Насосы/DB

DATA_BLOCK "Pump_1_DB"   // DB25
{ S7_Optimized_Access := 'FALSE' }
VERSION : 0.1
// stored: InstanceOfName Pump
"Pump"
BEGIN
END_DATA_BLOCK

DATA_BLOCK "Pump_2_DB"   // DB26
{ S7_Optimized_Access := 'FALSE' }
VERSION : 0.1
// stored: InstanceOfName Pump
"Pump"
BEGIN
END_DATA_BLOCK

// folder: (top level)

FUNCTION_BLOCK "Tank_Diarator"   // FB2, SCL
{ S7_Optimized_Access := 'TRUE' }
VERSION : 0.1
   VAR_INPUT
      bEnable : Bool;   // Разрешение на работу
      bPause : Bool;   // Остановка производства воды
      bReady_O2 : Bool;   // Готовность воды по датчику О2
      bControlO2_Type : Bool;   // 1 = по СО2, 0 по расходу. Тип контроля кол-ва кислорода (датчик, или расход)
      rPT01 : Real;   // Значение давления РТ01
      iРасход_Накопленный : Int;   // Значение накопленного расхода воды
      iFlow_SP : Int := 10;   // Уставка для Расхода по счетчику
      diTimeWaitingReadyO2 : DInt := 30;   // Времы выдержки до маркера готовности по датчику О2
   END_VAR
   VAR_OUTPUT
      bValve1 : Bool;   // Клапан набор
      bValve2 : Bool;   // Клапан регуллирующий, разрешение на работу
      bValve3 : Bool;   // Клапан слива в дренаж
      bValve5 : Bool;   // Клапан набора готовой воды в емкость
      bValve7 : Bool;   // Клапан СО2 в емкость подготовки
      bWaterReady : Bool;   // Маркер готовности воды
      bPump_1 : Bool;   // Разрешение на работу насоса
   END_VAR
   VAR RETAIN
      TON_ready_O2 : TON_TIME;   // Таймер готовности по датчику кислорода
   END_VAR
BEGIN
   //Перевод из мс в Сек для таймера ожидания О2
   #diTimeWaitingReadyO2 := #diTimeWaitingReadyO2 * 1000;

   //Начало если нет разрешения на работу
   IF NOT #bEnable THEN
       //Закрываем все клапана
       #bValve1 := #bValve2 := #bValve3 := #bValve5 := #bValve7 := FALSE;
       // Стоп насоса
       #bPump_1 := FALSE;
       //Нет работы сброс всего
       #bWaterReady := FALSE;
       #TON_ready_O2.IN := FALSE;
       RETURN;
   END_IF;

   //Начало работы блока если есть разрешение

   //Подача клапан 1
   IF #rPT01 >= "DB2_HMI_SET".rLewelTank1_Stop THEN
       #bValve1 := FALSE;
   ELSIF #rPT01 <= "DB2_HMI_SET".rLewelTank1_Start THEN
       #bValve1 := TRUE;
   END_IF;

   //#bValve1 := TRUE;   
   #bValve2 := TRUE;   //Регулятор расхода для емкости (ПИД разрешение работы)
   #bValve3 := TRUE;   //Слив воды в дренаж, пока вода не будет подготовлена
   #bValve7 := TRUE;   //Co2
   #bPump_1 := TRUE;   //Разрешение на работу ПИД насоса по датчику давления в емкости

   //Проверка выбора типа контроля уровня кислорода

   IF #bControlO2_Type THEN
       #TON_ready_O2(IN:= #bReady_O2, PT := #diTimeWaitingReadyO2, Q =>#bWaterReady);   //Время выдержки при достижении уставки по О2
   ELSE
       #bWaterReady := (#iРасход_Накопленный >= #iFlow_SP);
   END_IF;

   IF #bWaterReady THEN
       #bValve3 := FALSE;  //Слив в дренаж
       #bValve5 := TRUE;   //Подача воды в емкость
   ELSE
       #bValve3 := TRUE;  //Слив в дренаж
       #bValve5 := FALSE;   //Подача воды в емкость
   END_IF;

   IF #bPause THEN
       #bValve1 := #bValve2 := #bValve3 := #bValve5 := #bValve7 := FALSE;
       #bPump_1 := FALSE;
       //Нет работы сброс всего
       #bWaterReady := FALSE;
       //Сброс таймера
       #TON_ready_O2.IN := FALSE;
   END_IF;
END_FUNCTION_BLOCK

FUNCTION_BLOCK "FB_Control_O2"   // FB6, SCL
{ S7_Optimized_Access := 'TRUE' }
VERSION : 0.1
   VAR_INPUT
      bEnable : Bool;
      rO2_SP : Real;   // Уставка О2
      rO2_Actual : Real;   // Факт значение О2
      rGisteresis : Real;   // Гистерезис О2
      diTimeLost : DInt;   // Время за которое терпит отклонение от гистерезиса
   END_VAR
   VAR_OUTPUT
      bReady_O2 : Bool;
   END_VAR
   VAR
      UP_Limit : Real;
      DOWN_Limit : Real;
      bReady_Flag : Bool;
      TON_Lost_O2 : TON_TIME;
   END_VAR
BEGIN
   //Перевод значения в сек для таймера
   #diTimeLost := #diTimeLost * 1000;

   // Определение границ гистерезиса
   #UP_Limit := #rO2_SP + #rGisteresis;
   #DOWN_Limit := #rO2_SP - #rGisteresis;

   //Время ожидания для перехода в FALSE при выходе за уставку с учетом гистерезиса
   #TON_Lost_O2(IN := (#rO2_Actual >= #UP_Limit),
                PT := #diTimeLost);
   // Основная логика работы
   IF #TON_Lost_O2.Q THEN
       #bReady_Flag := FALSE;
   ELSIF #rO2_Actual >= #DOWN_Limit OR #rO2_Actual <= #UP_Limit THEN
       #bReady_Flag := TRUE;
   END_IF;

   IF NOT #bEnable THEN
       #bReady_Flag := FALSE;
   END_IF;

   #bReady_O2 := #bReady_Flag;
END_FUNCTION_BLOCK

FUNCTION_BLOCK "FB_Аварии"   // FB7, SCL
{ S7_Optimized_Access := 'FALSE' }
VERSION : 0.1
   VAR_INPUT
      Rtrig_Reset : Bool;
   END_VAR
   VAR_OUTPUT
      ALARM_Active : Bool;   // Флаг активной аварии
   END_VAR
   VAR
      LatchedEmergency : Bool;   // Зафиксированная аварийная ситуация
      bAlarmAvtomats : Bool;   // Авария автоматов
      bAlarmAI : Bool;   // Авария аналоговых датчиков
      bAlarmPumps : Bool;   // Авария насосов
      bAlarmConveyors : Bool;   // Авария Конвейеров
      bAlarmFVs : Bool;   // Авария клапанов
      bAlarmDI_all : Bool;   // Авария по дискретным входам "общая"
      bAlarmLowLevel : Bool;   // Авария по низкому уровню емкостей
      mReset : Bool;
      TON_LowLevel : TON_TIME;   // Таймер для аварийного уровня емкостей
      bResetaALARM : Bool;   // Сброс аварии (кнопка на панели/системе)
   END_VAR
   VAR_TEMP
      nAi : Int;
      nPump : Int;
      nConv : Int;
      nFV : Int;
      nAvtomat : Int;
      NumControlSensor : Int;
      numPump : Int;
   END_VAR
BEGIN
   REGION Предварительное отрицание
       // Сброс в 0 при отсутсвии аварий для цикла и массивов
       #bAlarmAvtomats := FALSE;
       #bAlarmAI := FALSE;
       #bAlarmPumps := FALSE;
       #bAlarmConveyors := FALSE;
       #bAlarmFVs := FALSE;


   END_REGION


   (*
   //Авария автоматические выключатели
   //--------------------------
   "Alarms".Avtomat_Off[1].ALARM  :=  "DI".DI_14.f_DI_out;
   "Alarms".Avtomat_Off[2].ALARM  :=  "DI".DI_16.f_DI_out;
   *)

   FOR #nAvtomat := 1 TO 2 DO
       IF "Alarms".Avtomat_Off[#nAvtomat].ALARM THEN
           #bAlarmAvtomats := TRUE;
       END_IF;
   END_FOR;

   //Авария аналоговых входов
   //
   //При выборе типа контроля готовности воды по счетчику - контроль датчика О2 - отключаем, если выбран контроль по датчику О2 - контролируем наличие аварии
   IF "bTypeControlO2" THEN
       #NumControlSensor := 7;     //Контролируем датчик О2 6 и 7 Ai вход
   ELSE
       #NumControlSensor := 5;
   END_IF;
   //--------------------------
   FOR #nAi := 1 TO #NumControlSensor DO
       IF "Alarms".Ai_Alarm[#nAi].ALARM THEN
           #bAlarmAI := TRUE;
       END_IF;
   END_FOR;

   //Авария НАСОСОВ
   //--------------------------

   FOR #nPump := 1 TO 5 DO
       IF "Alarms".Pump_Alarm[#nPump].ALARM THEN
           #bAlarmPumps := TRUE;
           #numPump := #nPump;

       END_IF;
   END_FOR;


   //Авария Клапанов
   //--------------------------

   FOR #nFV := 1 TO 10 DO
       IF "Alarms".FV_Alarm[#nFV].ALARM THEN
           #bAlarmFVs := TRUE;
       END_IF;
   END_FOR;



   //Авария по входам DI
   //---------------------------

   #bAlarmDI_all := "Alarms"."xE-Stop_1" OR
   "Alarms".xVoltRele OR
   "Alarms".xLongWaitWater OR "Alarms".xPressAir;


   //Обработка всех аварий с выводом сигнала наличия АВАРИЯ
   //----------------------------------------------------------------
                   IF #bAlarmAvtomats OR
                       #bAlarmAI OR
                       #bAlarmPumps OR
                       #bAlarmConveyors OR
                       #bAlarmFVs OR
                       #bAlarmDI_all OR
                       #bAlarmLowLevel
                   THEN

                       #ALARM_Active := TRUE;
                   END_IF;
     (*                     
   //Отлавливаем фронт Ресета....................................

   #bResetaALARM := #Rtrig_Reset AND NOT #mReset;
   #mReset := #Rtrig_Reset;
   *)

    //Если нужен жесткий сбро, игнорирует все аварии                      
   #bResetaALARM := #Rtrig_Reset;

   //-------------------------------------------------------------                       
                          // Сброс аварии
   IF #bResetaALARM THEN
       #ALARM_Active := FALSE;
   END_IF;
END_FUNCTION_BLOCK

FUNCTION_BLOCK "FB_Tank_2(Buffer)"   // FB8, SCL
{ S7_Optimized_Access := 'TRUE' }
VERSION : 0.1
   VAR_INPUT
      Enable : Bool;   // Разрешение
      bLSL02 : Bool;   // Нижний уровень
      bLSM03 : Bool;   // // Средний уровень
      bLSH04 : Bool;   // Верхний уровень
      tStartDelay : DInt;   // Время задержки пуска насоса после возврата уровня
      tNoWaterMax : DInt;   // сек, Максимальное время ожидания воды (для аварии)
      bResAlarm : Bool;   // Сброс аварий
   END_VAR
   VAR_OUTPUT
      bValve6 : Bool;   // Клапан раздачи воды
      bPump2Run : Bool;   // Насос P2
      bPause : Bool;   // Пауза (для остановки подачи воды в емкость)
      bAlarmNoWater : Bool;   // Авария — долго нет воды)
   END_VAR
   VAR
      tonStartDelay : TON_TIME;   // Таймер задержки старта
      tonNoWater : TON_TIME;   // Таймер отсутствия воды
      bStartPending : Bool;   // Флаг ожидания задержки
   END_VAR
BEGIN
   //Проверка разрешения на работу блока
   //....Сброс аварии...//
   IF #bResAlarm THEN
       // Уровень восстановился → сброс аварии и таймера "нет воды"
       #tonNoWater(IN := FALSE,
                   PT := t#0ms);
       #bAlarmNoWater := FALSE;
   END_IF;

   IF NOT #Enable THEN
       #bValve6 := FALSE;
       #bPump2Run := FALSE;
       #bPause := FALSE;
       //#bAlarmNoWater := FALSE;
       //Сброс таймеров
       #tonStartDelay(IN := FALSE, PT := t#0ms);
       #tonNoWater(IN := FALSE, PT := t#0ms);
       //Сброс метки ожидания
       #bStartPending := FALSE;
       RETURN;
   END_IF;

                   ///////////РАбота блока........\\\\\\\\\



   // ---------- Контроль верхнего уровня ----------
   IF #bLSH04 THEN
       #bPause := TRUE;   // ставим установку на паузу
   ELSIF NOT #bLSM03 THEN
       #bPause := FALSE;  // снимаем паузу
   END_IF;

   // ---------- Контроль нижнего уровня ----------
   IF NOT #bLSL02 THEN
       // Воды нет → стоп насос и клапан
       #bValve6 := FALSE;
       #bPump2Run := FALSE;

       // фиксируем, что после возврата LSL02 нужно выдержать паузу
       #bStartPending := TRUE;

       // запускаем таймер контроля отсутствия воды
       #tonNoWater(IN := TRUE,
                   PT := #tNoWaterMax * 1000);
       IF #tonNoWater.Q THEN
           #bAlarmNoWater := TRUE;
       END_IF;
   ELSE
       // Уровень восстановился → сброс аварии и таймера "нет воды"
       #tonNoWater(IN := FALSE,
                   PT := t#0ms);
       //#bAlarmNoWater := FALSE;

       IF #bStartPending THEN
           #tonStartDelay(IN := TRUE,
                          PT := #tStartDelay*1000);
           IF #tonStartDelay.Q THEN
               #bValve6 := TRUE;
               #bPump2Run := TRUE;
               #bStartPending := FALSE; // запуск выполнен
               #tonStartDelay(IN := FALSE, //сброс таймера задержки старта
                              PT := t#0ms);
           END_IF;
       ELSE
           // Уровень в норме, работаем
           #bValve6 := TRUE;
           #bPump2Run := TRUE;
       END_IF;
   END_IF;
END_FUNCTION_BLOCK

FUNCTION_BLOCK "FB_check_For_Start"   // FB9, SCL
{ S7_Optimized_Access := 'FALSE' }
VERSION : 0.1
   VAR_INPUT
      xHMI_Start : Bool;   // кнопка старта с HMI
      xEmergency_Stop : Bool;   // аварийный стоп
      xSystem_Ready : Bool;   // Готовность всех систем
      xStopHMI : Bool;   // Кнопка СТОП на HMI
   END_VAR
   VAR_OUTPUT
      xStart_Allowed : Bool;   // Разрешение на РАБОТУ
      xStart : Bool;   // Работа пастеризатора
   END_VAR
   VAR
      "m" : Bool;   // memory
   END_VAR
BEGIN

   //Проверка на разрешение работы.
   //
   IF NOT #xEmergency_Stop AND #xSystem_Ready THEN
       #xStart_Allowed := TRUE;
   ELSE
       #xStart_Allowed := FALSE;
   END_IF;

   #xStart := (#xStart OR #xHMI_Start) AND NOT (#xEmergency_Stop OR #xStopHMI);
END_FUNCTION_BLOCK

FUNCTION_BLOCK "FB_Control_Press_Tank2"   // FB10, SCL
{ S7_Optimized_Access := 'TRUE' }
VERSION : 0.1
   VAR_INPUT
      Enable : Bool;   // Разрешение работы
      rPT02 : Real;   // Давление в емкости 2 (фактическое)
      rPT02_SP : Real;   // Уставка давления
      tOpenDelay : DInt;   // Задержка на открытие клапана 9
      tCloseDelay : DInt;   // Задержка на закрытие клапана 9
   END_VAR
   VAR_OUTPUT
      bValve9 : Bool;   // Управление клапаном 9
   END_VAR
   VAR
      tonOpenDelay : TON_TIME;   // Таймер задержки открытия
      tonCloseDelay : TON_TIME;   // Таймер задержки закрытия
      bRequestOpen : Bool;   // Запрос открыть
      bRequestClose : Bool;   // Запрос закрыть
   END_VAR
BEGIN
   #tOpenDelay := #tOpenDelay * 1000;
   #tCloseDelay := #tCloseDelay * 1000;
   //Проверка разрешения на работу блока

   IF NOT #Enable THEN
       #bValve9 := FALSE;
       #tonOpenDelay(IN := FALSE,
                     PT := t#0ms);
       #tonCloseDelay(IN := FALSE,
                      PT := t#0ms);
       #bRequestOpen := FALSE;
       #bRequestClose := FALSE;
       RETURN;
   END_IF;

   // --- Условия ---
   #bRequestOpen := (#rPT02 < #rPT02_SP);   // давление ниже нормы
   #bRequestClose := (#rPT02 >= #rPT02_SP);  // давление достигло нормы

   // --- Логика открытия ---
   IF #bRequestOpen THEN
       #tonOpenDelay(IN := TRUE,
                     PT := #tOpenDelay);
       #tonCloseDelay(IN := FALSE,
                      PT := t#0ms);

       IF #tonOpenDelay.Q THEN
           #bValve9 := TRUE;
       END_IF;
   ELSE
       #tonOpenDelay(IN := FALSE,
                     PT := t#0ms);
   END_IF;

   // --- Логика закрытия ---
   IF #bRequestClose THEN
       #tonCloseDelay(IN := TRUE,
                      PT := #tCloseDelay);
       #tonOpenDelay(IN := FALSE,
                     PT := t#0ms);

       IF #tonCloseDelay.Q THEN
           #bValve9 := FALSE;
       END_IF;
   ELSE
       #tonCloseDelay(IN := FALSE,
                      PT := t#0ms);
   END_IF;
END_FUNCTION_BLOCK

FUNCTION_BLOCK "FB_CIP"   // FB11, SCL
{ S7_Optimized_Access := 'TRUE' }
VERSION : 0.1
   VAR_INPUT
      Enable : Bool;   // Разрешение
      tFlipTime : DInt;   // Время переключения клапанов 8-10-5
      tFlipPause : DInt;   // Выдержка после полного цикла
      "СенсорТанк-1" : Real;
   END_VAR
   VAR_OUTPUT
      bValve1 : Bool;
      bValve2 : Bool;
      bValve4 : Bool;
      bValve6 : Bool;
      bValve5 : Bool;
      bValve8 : Bool;
      bValve10 : Bool;
      bPump1 : Bool;
      bPump2 : Bool;
   END_VAR
   VAR
      tonFlip : TON_TIME;   // таймер для переключений внутри цикла
      tonPause : TON_TIME;   // таймер паузы после цикла
      iFlipStep : Int;
      bInPause : Bool;
   END_VAR
BEGIN
   //Перевод времени для таймеров в сек
   #tFlipTime := #tFlipTime * 1000;
   #tFlipPause := #tFlipPause * 1000;

   IF NOT #Enable THEN
       #bValve1 := FALSE;
       #bValve2 := FALSE;
       #bValve4 := FALSE;
       #bValve5 := FALSE;
       #bValve6 := FALSE;
       #bValve8 := FALSE;
       #bValve10 := FALSE;
       #bPump1 := FALSE;
       #bPump2 := FALSE;

       #tonFlip(IN := FALSE,
                PT := t#0ms);
       #tonPause(IN := FALSE,
                 PT := t#0ms);
       #iFlipStep := 0;
       #bInPause := FALSE;
       RETURN;
   END_IF;

   // --- Постоянные включения ---
   //Подача клапан 1
   IF #"СенсорТанк-1" >= 95.0 THEN
       #bValve1 := FALSE;
   ELSIF #"СенсорТанк-1" <= 90.0 THEN
       #bValve1 := TRUE;
   END_IF;

   #bValve2 := TRUE;
   #bValve4 := TRUE;
   #bValve6 := TRUE;

   #bPump1 := TRUE;
   #bPump2 := TRUE;


   // --- Флоппинг ---
   IF NOT #bInPause THEN
       #tonFlip(IN := TRUE,
                PT := #tFlipTime);

       IF #tonFlip.Q THEN
           #tonFlip(IN := FALSE, PT := t#0ms);
           #iFlipStep := #iFlipStep + 1;

           IF #iFlipStep > 3 THEN
               // отработали все три шага → переходим в паузу
               #iFlipStep := 0;
               #bInPause := TRUE;
               #tonPause(IN := TRUE,
                         PT := #tFlipPause);
           END_IF;
       END_IF;
   ELSE
       // Пауза после цикла
       #tonPause(IN := TRUE,
                 PT := #tFlipPause);
       IF #tonPause.Q THEN
           #tonPause(IN := FALSE,
                     PT := t#0ms);
           #bInPause := FALSE;
           #iFlipStep := 1; // начинаем новый цикл с клапана 8
       END_IF;
   END_IF;

   // Управление клапанами по шагам
   CASE #iFlipStep OF
       1: // Открыт клапан 8
           #bValve8 := TRUE;
           #bValve10 := FALSE;
           #bValve5 := FALSE;
       2: // Открыт клапан 10
           #bValve8 := FALSE;
           #bValve10 := TRUE;
           #bValve5 := FALSE;
       3: // Открыт клапан 5
           #bValve8 := FALSE;
           #bValve10 := FALSE;
           #bValve5 := TRUE;
       ELSE
           // пауза или IDLE
           #bValve8 := FALSE;
           #bValve10 := FALSE;
           #bValve5 := FALSE;
   END_CASE;
END_FUNCTION_BLOCK

FUNCTION_BLOCK "FB_OwerPress_Tank_2"   // FB18, SCL
{ S7_Optimized_Access := 'FALSE' }
VERSION : 0.1
   VAR_INPUT
      bEn : Bool;   // Разрешение работы блока
      rPressSensor : Real;   // Значение датчика давления
      rSetOwerPress : Real;   // Уставка давления для сброса
      rSetHisteresis : Real;   // Уставка гистерезиса
   END_VAR
   VAR_OUTPUT
      bValve : Bool;   // Выход на клапан
      bHisUp : Real;
      bHisDown : Real;
   END_VAR
   VAR
      b_ActualOut : Bool;   // Внутреняя переменная для выхода
      fb_HisterPress : "fb_Histeresis";
   END_VAR
BEGIN
   //Разрешение работать блоку контроля давления
   IF NOT #bEn THEN
       #b_ActualOut := FALSE;
       #bValve := FALSE;
       RETURN;
   END_IF;

   #fb_HisterPress(bEnable:=TRUE,
                   rInputValue:=#rPressSensor,
                   rSetpoint:=#rSetOwerPress,
                   rUpperHyst:=#rSetHisteresis,
                   rLowerHyst:=#rSetHisteresis,
                   bOutput=>#b_ActualOut,
                   rUpperThreshold=>#bHisUp,
                   rLowerThreshold=>#bHisDown);

   #bValve := #b_ActualOut;
END_FUNCTION_BLOCK

FUNCTION_BLOCK "FB_SVETOFOR"   // FB19, SCL
{ S7_Optimized_Access := 'TRUE' }
VERSION : 0.1
   VAR_OUTPUT
      Зеленый : Bool;   // Включение зеленого света
      Желтый : Bool;   // Включение желтого
      Красный : Bool;   // красного
      Пищалка : Bool;
   END_VAR
   VAR
      AlarmPress : Bool;   // Авария по давлению
      rTrig_Alarm : "R_trig";   // Фронт аварии
   END_VAR
BEGIN
   //Включение зеленого при старте конвейеров
   //
   IF "bStartWork_Main" THEN
       #Зеленый := TRUE;
   ELSIF "bStartWork_Main" AND NOT "Разрешение работы конвейера" THEN
       #Зеленый := "Time_2s";
   ELSE
       #Зеленый := FALSE;
   END_IF;

   // Упрвавление желтым сигналом
   // 
   IF "bStartWork_Main" AND "bPosition_Diarator" AND  NOT "bDiarator_WaterReady" THEN
       #Желтый := TRUE;
   ELSE
       #Желтый := FALSE;
   END_IF;




   //Управление карасным сигналом
   //
   #Красный := FALSE;
   IF "bMain_AlarmSystem" THEN
       #Красный := TRUE;
   END_IF;

   #rTrig_Alarm(In := "bMain_AlarmSystem");

   // Управление пищалкой
   // 
   IF (#Пищалка OR #rTrig_Alarm.Q) AND NOT "bZoomerOff" THEN
       #Пищалка := TRUE;

   ELSIF "bStartWork_Main" AND "bOpenWindStartConveyor" THEN
       #Пищалка := "Time_1s";
   ELSE
       #Пищалка := FALSE;

   END_IF;

   "R_trig_DB_Pause"(In:=("iHMI_Num_StatrPaster" = 40));


   // Включение пищалки если режим ПАУЗА
   IF "R_trig_DB_Pause".Q THEN
       #Пищалка := TRUE;
   END_IF;

   IF "bZoomerOff" THEN
       #Пищалка := FALSE;
   END_IF;
END_FUNCTION_BLOCK

FUNCTION "Клапана_О/З" : Void   // FC1, LAD
{ S7_Optimized_Access := 'TRUE' }
VERSION : 0.1
BEGIN

REGION Network 1: FV-1
   // Регулирующий клапан Преднагрев
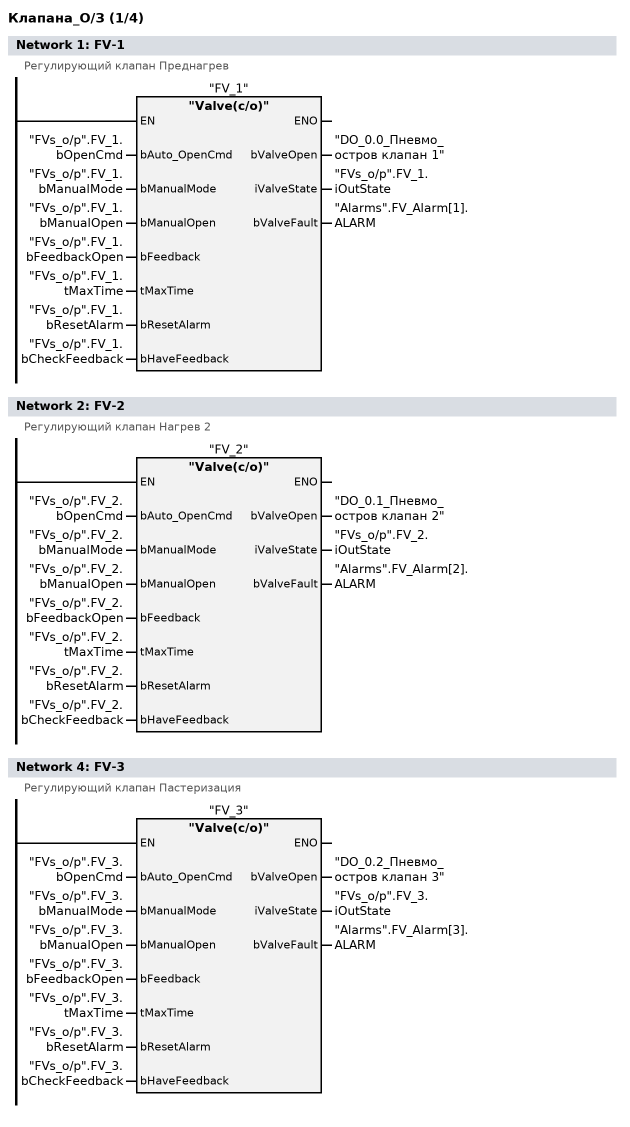
   RUNG wire#powerrail
      "FV_1"(bAuto_OpenCmd := "FVs_o/p".FV_1.bOpenCmd, bManualMode := "FVs_o/p".FV_1.bManualMode, bManualOpen := "FVs_o/p".FV_1.bManualOpen, bFeedback := "FVs_o/p".FV_1.bFeedbackOpen, tMaxTime := "FVs_o/p".FV_1.tMaxTime, bResetAlarm := "FVs_o/p".FV_1.bResetAlarm, bHaveFeedback := "FVs_o/p".FV_1.bCheckFeedback, bValveOpen => "DO_0.0_Пневмо_остров клапан 1", iValveState => "FVs_o/p".FV_1.iOutState, bValveFault => "Alarms".FV_Alarm[1].ALARM)
   END_RUNG
   // the same network as SCL:
   "FV_1"(bAuto_OpenCmd := "FVs_o/p".FV_1.bOpenCmd,   // "Valve(c/o)"
          bManualMode := "FVs_o/p".FV_1.bManualMode,
          bManualOpen := "FVs_o/p".FV_1.bManualOpen,
          bFeedback := "FVs_o/p".FV_1.bFeedbackOpen,
          tMaxTime := "FVs_o/p".FV_1.tMaxTime,
          bResetAlarm := "FVs_o/p".FV_1.bResetAlarm,
          bHaveFeedback := "FVs_o/p".FV_1.bCheckFeedback,
          bValveOpen => "DO_0.0_Пневмо_остров клапан 1",
          iValveState => "FVs_o/p".FV_1.iOutState,
          bValveFault => "Alarms".FV_Alarm[1].ALARM);
END_REGION

REGION Network 2: FV-2
   // Регулирующий клапан Нагрев 2
   RUNG wire#powerrail
      "FV_2"(bAuto_OpenCmd := "FVs_o/p".FV_2.bOpenCmd, bManualMode := "FVs_o/p".FV_2.bManualMode, bManualOpen := "FVs_o/p".FV_2.bManualOpen, bFeedback := "FVs_o/p".FV_2.bFeedbackOpen, tMaxTime := "FVs_o/p".FV_2.tMaxTime, bResetAlarm := "FVs_o/p".FV_2.bResetAlarm, bHaveFeedback := "FVs_o/p".FV_2.bCheckFeedback, bValveOpen => "DO_0.1_Пневмо_остров клапан 2", iValveState => "FVs_o/p".FV_2.iOutState, bValveFault => "Alarms".FV_Alarm[2].ALARM)
   END_RUNG
   // the same network as SCL:
   "FV_2"(bAuto_OpenCmd := "FVs_o/p".FV_2.bOpenCmd,   // "Valve(c/o)"
          bManualMode := "FVs_o/p".FV_2.bManualMode,
          bManualOpen := "FVs_o/p".FV_2.bManualOpen,
          bFeedback := "FVs_o/p".FV_2.bFeedbackOpen,
          tMaxTime := "FVs_o/p".FV_2.tMaxTime,
          bResetAlarm := "FVs_o/p".FV_2.bResetAlarm,
          bHaveFeedback := "FVs_o/p".FV_2.bCheckFeedback,
          bValveOpen => "DO_0.1_Пневмо_остров клапан 2",
          iValveState => "FVs_o/p".FV_2.iOutState,
          bValveFault => "Alarms".FV_Alarm[2].ALARM);
END_REGION

REGION Network 3 (SCL): DO - регул клапан
   // Специфика регулятора
   "DO_0.1_Пневмо_остров клапан 2" := true;
END_REGION

REGION Network 4: FV-3
   // Регулирующий клапан Пастеризация
   RUNG wire#powerrail
      "FV_3"(bAuto_OpenCmd := "FVs_o/p".FV_3.bOpenCmd, bManualMode := "FVs_o/p".FV_3.bManualMode, bManualOpen := "FVs_o/p".FV_3.bManualOpen, bFeedback := "FVs_o/p".FV_3.bFeedbackOpen, tMaxTime := "FVs_o/p".FV_3.tMaxTime, bResetAlarm := "FVs_o/p".FV_3.bResetAlarm, bHaveFeedback := "FVs_o/p".FV_3.bCheckFeedback, bValveOpen => "DO_0.2_Пневмо_остров клапан 3", iValveState => "FVs_o/p".FV_3.iOutState, bValveFault => "Alarms".FV_Alarm[3].ALARM)
   END_RUNG
   // the same network as SCL:
   "FV_3"(bAuto_OpenCmd := "FVs_o/p".FV_3.bOpenCmd,   // "Valve(c/o)"
          bManualMode := "FVs_o/p".FV_3.bManualMode,
          bManualOpen := "FVs_o/p".FV_3.bManualOpen,
          bFeedback := "FVs_o/p".FV_3.bFeedbackOpen,
          tMaxTime := "FVs_o/p".FV_3.tMaxTime,
          bResetAlarm := "FVs_o/p".FV_3.bResetAlarm,
          bHaveFeedback := "FVs_o/p".FV_3.bCheckFeedback,
          bValveOpen => "DO_0.2_Пневмо_остров клапан 3",
          iValveState => "FVs_o/p".FV_3.iOutState,
          bValveFault => "Alarms".FV_Alarm[3].ALARM);
END_REGION

REGION Network 5: FV-4
   // Регулирующий клапан Охлаждения - 2
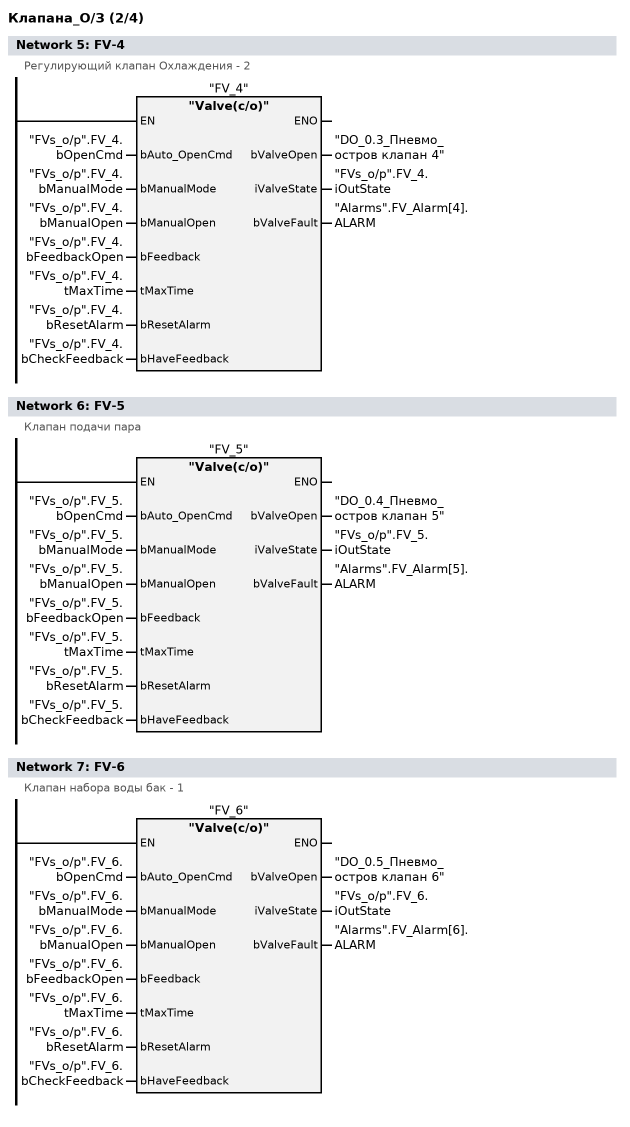
   RUNG wire#powerrail
      "FV_4"(bAuto_OpenCmd := "FVs_o/p".FV_4.bOpenCmd, bManualMode := "FVs_o/p".FV_4.bManualMode, bManualOpen := "FVs_o/p".FV_4.bManualOpen, bFeedback := "FVs_o/p".FV_4.bFeedbackOpen, tMaxTime := "FVs_o/p".FV_4.tMaxTime, bResetAlarm := "FVs_o/p".FV_4.bResetAlarm, bHaveFeedback := "FVs_o/p".FV_4.bCheckFeedback, bValveOpen => "DO_0.3_Пневмо_остров клапан 4", iValveState => "FVs_o/p".FV_4.iOutState, bValveFault => "Alarms".FV_Alarm[4].ALARM)
   END_RUNG
   // the same network as SCL:
   "FV_4"(bAuto_OpenCmd := "FVs_o/p".FV_4.bOpenCmd,   // "Valve(c/o)"
          bManualMode := "FVs_o/p".FV_4.bManualMode,
          bManualOpen := "FVs_o/p".FV_4.bManualOpen,
          bFeedback := "FVs_o/p".FV_4.bFeedbackOpen,
          tMaxTime := "FVs_o/p".FV_4.tMaxTime,
          bResetAlarm := "FVs_o/p".FV_4.bResetAlarm,
          bHaveFeedback := "FVs_o/p".FV_4.bCheckFeedback,
          bValveOpen => "DO_0.3_Пневмо_остров клапан 4",
          iValveState => "FVs_o/p".FV_4.iOutState,
          bValveFault => "Alarms".FV_Alarm[4].ALARM);
END_REGION

REGION Network 6: FV-5
   // Клапан подачи пара
   RUNG wire#powerrail
      "FV_5"(bAuto_OpenCmd := "FVs_o/p".FV_5.bOpenCmd, bManualMode := "FVs_o/p".FV_5.bManualMode, bManualOpen := "FVs_o/p".FV_5.bManualOpen, bFeedback := "FVs_o/p".FV_5.bFeedbackOpen, tMaxTime := "FVs_o/p".FV_5.tMaxTime, bResetAlarm := "FVs_o/p".FV_5.bResetAlarm, bHaveFeedback := "FVs_o/p".FV_5.bCheckFeedback, bValveOpen => "DO_0.4_Пневмо_остров клапан 5", iValveState => "FVs_o/p".FV_5.iOutState, bValveFault => "Alarms".FV_Alarm[5].ALARM)
   END_RUNG
   // the same network as SCL:
   "FV_5"(bAuto_OpenCmd := "FVs_o/p".FV_5.bOpenCmd,   // "Valve(c/o)"
          bManualMode := "FVs_o/p".FV_5.bManualMode,
          bManualOpen := "FVs_o/p".FV_5.bManualOpen,
          bFeedback := "FVs_o/p".FV_5.bFeedbackOpen,
          tMaxTime := "FVs_o/p".FV_5.tMaxTime,
          bResetAlarm := "FVs_o/p".FV_5.bResetAlarm,
          bHaveFeedback := "FVs_o/p".FV_5.bCheckFeedback,
          bValveOpen => "DO_0.4_Пневмо_остров клапан 5",
          iValveState => "FVs_o/p".FV_5.iOutState,
          bValveFault => "Alarms".FV_Alarm[5].ALARM);
END_REGION

REGION Network 7: FV-6
   // Клапан набора воды бак - 1
   RUNG wire#powerrail
      "FV_6"(bAuto_OpenCmd := "FVs_o/p".FV_6.bOpenCmd, bManualMode := "FVs_o/p".FV_6.bManualMode, bManualOpen := "FVs_o/p".FV_6.bManualOpen, bFeedback := "FVs_o/p".FV_6.bFeedbackOpen, tMaxTime := "FVs_o/p".FV_6.tMaxTime, bResetAlarm := "FVs_o/p".FV_6.bResetAlarm, bHaveFeedback := "FVs_o/p".FV_6.bCheckFeedback, bValveOpen => "DO_0.5_Пневмо_остров клапан 6", iValveState => "FVs_o/p".FV_6.iOutState, bValveFault => "Alarms".FV_Alarm[6].ALARM)
   END_RUNG
   // the same network as SCL:
   "FV_6"(bAuto_OpenCmd := "FVs_o/p".FV_6.bOpenCmd,   // "Valve(c/o)"
          bManualMode := "FVs_o/p".FV_6.bManualMode,
          bManualOpen := "FVs_o/p".FV_6.bManualOpen,
          bFeedback := "FVs_o/p".FV_6.bFeedbackOpen,
          tMaxTime := "FVs_o/p".FV_6.tMaxTime,
          bResetAlarm := "FVs_o/p".FV_6.bResetAlarm,
          bHaveFeedback := "FVs_o/p".FV_6.bCheckFeedback,
          bValveOpen => "DO_0.5_Пневмо_остров клапан 6",
          iValveState => "FVs_o/p".FV_6.iOutState,
          bValveFault => "Alarms".FV_Alarm[6].ALARM);
END_REGION

REGION Network 8: FV-7
   // Клапан набора воды бак - 2
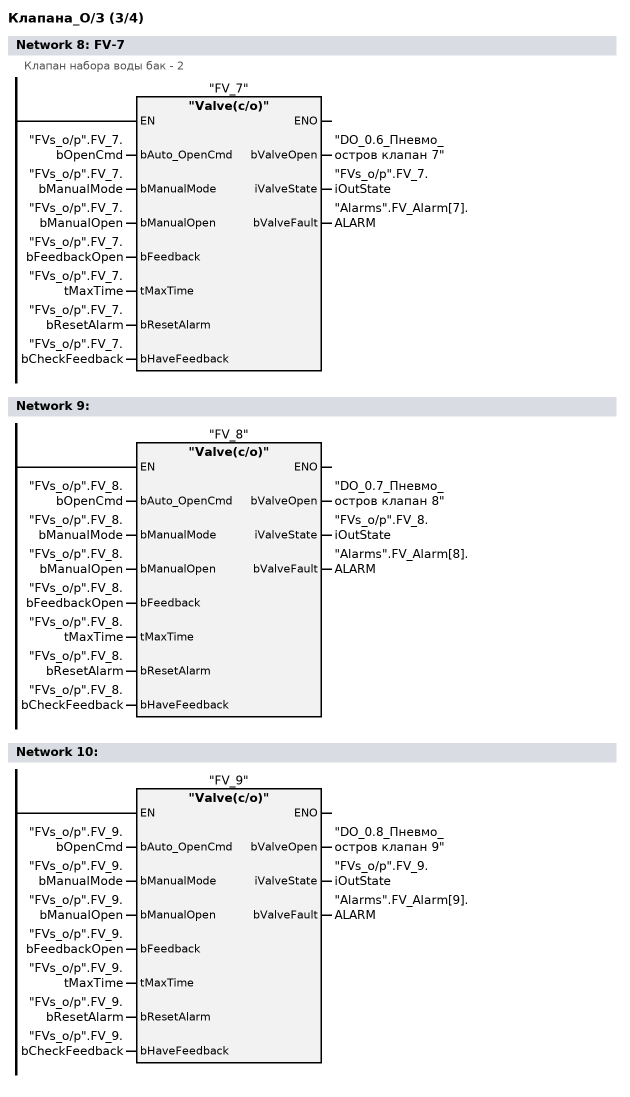
   RUNG wire#powerrail
      "FV_7"(bAuto_OpenCmd := "FVs_o/p".FV_7.bOpenCmd, bManualMode := "FVs_o/p".FV_7.bManualMode, bManualOpen := "FVs_o/p".FV_7.bManualOpen, bFeedback := "FVs_o/p".FV_7.bFeedbackOpen, tMaxTime := "FVs_o/p".FV_7.tMaxTime, bResetAlarm := "FVs_o/p".FV_7.bResetAlarm, bHaveFeedback := "FVs_o/p".FV_7.bCheckFeedback, bValveOpen => "DO_0.6_Пневмо_остров клапан 7", iValveState => "FVs_o/p".FV_7.iOutState, bValveFault => "Alarms".FV_Alarm[7].ALARM)
   END_RUNG
   // the same network as SCL:
   "FV_7"(bAuto_OpenCmd := "FVs_o/p".FV_7.bOpenCmd,   // "Valve(c/o)"
          bManualMode := "FVs_o/p".FV_7.bManualMode,
          bManualOpen := "FVs_o/p".FV_7.bManualOpen,
          bFeedback := "FVs_o/p".FV_7.bFeedbackOpen,
          tMaxTime := "FVs_o/p".FV_7.tMaxTime,
          bResetAlarm := "FVs_o/p".FV_7.bResetAlarm,
          bHaveFeedback := "FVs_o/p".FV_7.bCheckFeedback,
          bValveOpen => "DO_0.6_Пневмо_остров клапан 7",
          iValveState => "FVs_o/p".FV_7.iOutState,
          bValveFault => "Alarms".FV_Alarm[7].ALARM);
END_REGION

REGION Network 9
   RUNG wire#powerrail
      "FV_8"(bAuto_OpenCmd := "FVs_o/p".FV_8.bOpenCmd, bManualMode := "FVs_o/p".FV_8.bManualMode, bManualOpen := "FVs_o/p".FV_8.bManualOpen, bFeedback := "FVs_o/p".FV_8.bFeedbackOpen, tMaxTime := "FVs_o/p".FV_8.tMaxTime, bResetAlarm := "FVs_o/p".FV_8.bResetAlarm, bHaveFeedback := "FVs_o/p".FV_8.bCheckFeedback, bValveOpen => "DO_0.7_Пневмо_остров клапан 8", iValveState => "FVs_o/p".FV_8.iOutState, bValveFault => "Alarms".FV_Alarm[8].ALARM)
   END_RUNG
   // the same network as SCL:
   "FV_8"(bAuto_OpenCmd := "FVs_o/p".FV_8.bOpenCmd,   // "Valve(c/o)"
          bManualMode := "FVs_o/p".FV_8.bManualMode,
          bManualOpen := "FVs_o/p".FV_8.bManualOpen,
          bFeedback := "FVs_o/p".FV_8.bFeedbackOpen,
          tMaxTime := "FVs_o/p".FV_8.tMaxTime,
          bResetAlarm := "FVs_o/p".FV_8.bResetAlarm,
          bHaveFeedback := "FVs_o/p".FV_8.bCheckFeedback,
          bValveOpen => "DO_0.7_Пневмо_остров клапан 8",
          iValveState => "FVs_o/p".FV_8.iOutState,
          bValveFault => "Alarms".FV_Alarm[8].ALARM);
END_REGION

REGION Network 10
   RUNG wire#powerrail
      "FV_9"(bAuto_OpenCmd := "FVs_o/p".FV_9.bOpenCmd, bManualMode := "FVs_o/p".FV_9.bManualMode, bManualOpen := "FVs_o/p".FV_9.bManualOpen, bFeedback := "FVs_o/p".FV_9.bFeedbackOpen, tMaxTime := "FVs_o/p".FV_9.tMaxTime, bResetAlarm := "FVs_o/p".FV_9.bResetAlarm, bHaveFeedback := "FVs_o/p".FV_9.bCheckFeedback, bValveOpen => "DO_0.8_Пневмо_остров клапан 9", iValveState => "FVs_o/p".FV_9.iOutState, bValveFault => "Alarms".FV_Alarm[9].ALARM)
   END_RUNG
   // the same network as SCL:
   "FV_9"(bAuto_OpenCmd := "FVs_o/p".FV_9.bOpenCmd,   // "Valve(c/o)"
          bManualMode := "FVs_o/p".FV_9.bManualMode,
          bManualOpen := "FVs_o/p".FV_9.bManualOpen,
          bFeedback := "FVs_o/p".FV_9.bFeedbackOpen,
          tMaxTime := "FVs_o/p".FV_9.tMaxTime,
          bResetAlarm := "FVs_o/p".FV_9.bResetAlarm,
          bHaveFeedback := "FVs_o/p".FV_9.bCheckFeedback,
          bValveOpen => "DO_0.8_Пневмо_остров клапан 9",
          iValveState => "FVs_o/p".FV_9.iOutState,
          bValveFault => "Alarms".FV_Alarm[9].ALARM);
END_REGION

REGION Network 11
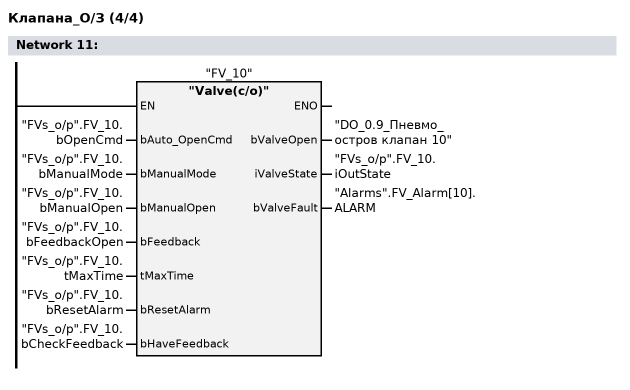
   RUNG wire#powerrail
      "FV_10"(bAuto_OpenCmd := "FVs_o/p".FV_10.bOpenCmd, bManualMode := "FVs_o/p".FV_10.bManualMode, bManualOpen := "FVs_o/p".FV_10.bManualOpen, bFeedback := "FVs_o/p".FV_10.bFeedbackOpen, tMaxTime := "FVs_o/p".FV_10.tMaxTime, bResetAlarm := "FVs_o/p".FV_10.bResetAlarm, bHaveFeedback := "FVs_o/p".FV_10.bCheckFeedback, bValveOpen => "DO_0.9_Пневмо_остров клапан 10", iValveState => "FVs_o/p".FV_10.iOutState, bValveFault => "Alarms".FV_Alarm[10].ALARM)
   END_RUNG
   // the same network as SCL:
   "FV_10"(bAuto_OpenCmd := "FVs_o/p".FV_10.bOpenCmd,   // "Valve(c/o)"
           bManualMode := "FVs_o/p".FV_10.bManualMode,
           bManualOpen := "FVs_o/p".FV_10.bManualOpen,
           bFeedback := "FVs_o/p".FV_10.bFeedbackOpen,
           tMaxTime := "FVs_o/p".FV_10.tMaxTime,
           bResetAlarm := "FVs_o/p".FV_10.bResetAlarm,
           bHaveFeedback := "FVs_o/p".FV_10.bCheckFeedback,
           bValveOpen => "DO_0.9_Пневмо_остров клапан 10",
           iValveState => "FVs_o/p".FV_10.iOutState,
           bValveFault => "Alarms".FV_Alarm[10].ALARM);
END_REGION
END_FUNCTION

FUNCTION "Клапана_Регул" : Void   // FC2, LAD
{ S7_Optimized_Access := 'TRUE' }
VERSION : 0.1
BEGIN

REGION Network 1: Клапан 2
   // Клапан с регурировкой потока
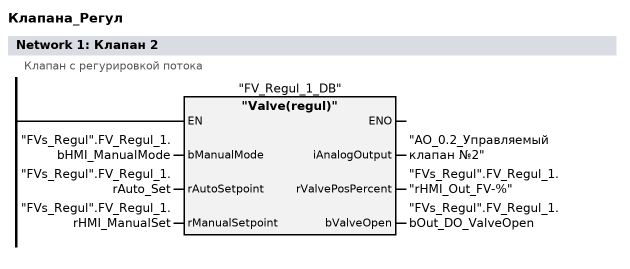
   RUNG wire#powerrail
      "FV_Regul_1_DB"(bManualMode := "FVs_Regul".FV_Regul_1.bHMI_ManualMode, rAutoSetpoint := "FVs_Regul".FV_Regul_1.rAuto_Set, rManualSetpoint := "FVs_Regul".FV_Regul_1.rHMI_ManualSet, iAnalogOutput => "AO_0.2_Управляемый клапан №2", rValvePosPercent => "FVs_Regul".FV_Regul_1."rHMI_Out_FV-%", bValveOpen => "FVs_Regul".FV_Regul_1.bOut_DO_ValveOpen)
   END_RUNG
   // the same network as SCL:
   "FV_Regul_1_DB"(bManualMode := "FVs_Regul".FV_Regul_1.bHMI_ManualMode,   // "Valve(regul)"
                   rAutoSetpoint := "FVs_Regul".FV_Regul_1.rAuto_Set,
                   rManualSetpoint := "FVs_Regul".FV_Regul_1.rHMI_ManualSet,
                   iAnalogOutput => "AO_0.2_Управляемый клапан №2",
                   rValvePosPercent => "FVs_Regul".FV_Regul_1."rHMI_Out_FV-%",
                   bValveOpen => "FVs_Regul".FV_Regul_1.bOut_DO_ValveOpen);
END_REGION

REGION Network 2 (SCL): Клапана регулирующие ручной режим с вфходом DO
   // Для перевода клапана регулирующего в ручной режим должен перейти по сигналу от ручного режим с клапана DO, т.е. для работы клапана регулирующего необходим сигнал DO
   "FVs_o/p".FV_2.bManualMode := "FVs_Regul".FV_Regul_1.bHMI_ManualMode;
END_REGION
END_FUNCTION

FUNCTION "FC_STOP1" : Void   // FC3, SCL
{ S7_Optimized_Access := 'TRUE' }
VERSION : 0.1
   VAR_INPUT
      Not_Start : Bool;
   END_VAR
BEGIN
   IF #Not_Start THEN
       //Закрыть клапана
       "FVs_o/p".FV_1.bOpenCmd := FALSE;
       "FVs_o/p".FV_2.bOpenCmd := FALSE;
       "FVs_o/p".FV_3.bOpenCmd := FALSE;
       "FVs_o/p".FV_4.bOpenCmd := FALSE;
       "FVs_o/p".FV_5.bOpenCmd := FALSE;
       "FVs_o/p".FV_6.bOpenCmd := FALSE;
       "FVs_o/p".FV_7.bOpenCmd := FALSE;
       "FVs_o/p".FV_8.bOpenCmd := FALSE;
       "FVs_o/p".FV_9.bOpenCmd := FALSE;
      // "FVs_o/p".FV_10.bOpenCmd := FALSE;

      // Остановить "Насосы"
       "Pumps".Pump_1.bAutoStartPump := FALSE;
       "Pumps".Pump_2.bAutoStartPump := FALSE;
       "Pumps".Pump_1.rAutoSpeedPump := 0.0;
       "Pumps".Pump_2.rAutoSpeedPump := 0.0;
   END_IF;

   //       .................СИП.....................
   // если режим СИП то закрываем клапана с задержкой для слива в канализацию
   IF "bPosition_CIP" THEN
       IF "R_trig_DB_Stop_CIP".Q THEN
           "m_STOP" := TRUE;
       END_IF;

   //........Управляю клапанами от таймера с задержкой для сброса в дренаж ...........
       IF "m_STOP" THEN
           "FVs_o/p".FV_3.bOpenCmd := NOT "_bCloseFV_CIP"; //Управляющий сигнал таймера (см. начало)
           "FVs_o/p".FV_8.bOpenCmd := NOT "_bCloseFV_CIP";
           "FVs_o/p".FV_10.bOpenCmd := NOT "_bCloseFV_CIP";
       END_IF;
    //.....Сброс таймера....   
       IF "_bCloseFV_CIP" THEN
           "m_STOP" := FALSE;
       END_IF;

   END_IF;
END_FUNCTION

FUNCTION "Аварии/res" : Void   // FC4, LAD
{ S7_Optimized_Access := 'TRUE' }
VERSION : 0.1
   VAR_INPUT
      bResrt : Bool;
   END_VAR
   VAR_OUTPUT
      xAlarm : Bool;   // Есть активные аварии
   END_VAR
BEGIN

REGION Network 1
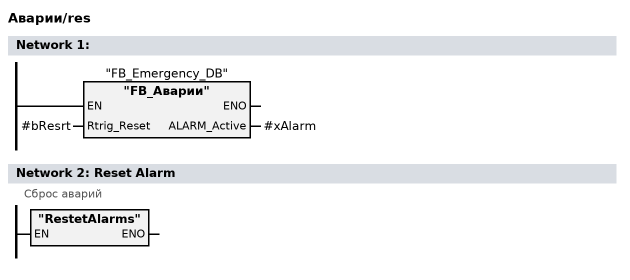
   RUNG wire#powerrail
      "FB_Emergency_DB"(Rtrig_Reset := #bResrt, ALARM_Active => #xAlarm)
   END_RUNG
   // the same network as SCL:
   "FB_Emergency_DB"(Rtrig_Reset := #bResrt, ALARM_Active => #xAlarm);   // "FB_Аварии"
END_REGION

REGION Network 2: Reset Alarm
   // Сброс аварий
   RUNG wire#powerrail
      "RestetAlarms"()
   END_RUNG
   // the same network as SCL:
   "RestetAlarms"();
END_REGION

REGION Network 3 (SCL): Есть активные аварии
END_REGION
END_FUNCTION

FUNCTION "Насосы" : Void   // FC5, LAD
{ S7_Optimized_Access := 'TRUE' }
VERSION : 0.1
// Блоки управления Насосами
BEGIN

REGION Network 1: Насос 1
   // Привязать датчик давления с уставкой для контроля сухого хода
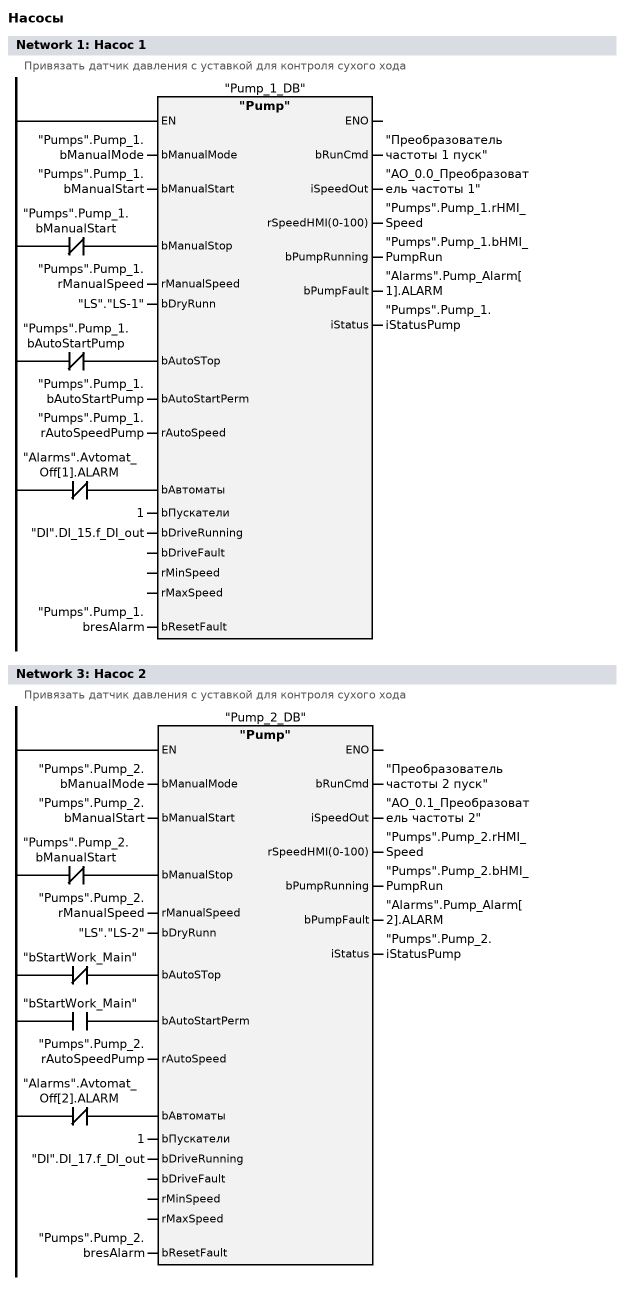
   RUNG wire#powerrail
      "Pump_1_DB"(bManualStop := wire#w1, bAutoSTop := wire#w2, bАвтоматы := wire#w3, bManualMode := "Pumps".Pump_1.bManualMode, bManualStart := "Pumps".Pump_1.bManualStart, rManualSpeed := "Pumps".Pump_1.rManualSpeed, bDryRunn := "LS"."LS-1", bAutoStartPerm := "Pumps".Pump_1.bAutoStartPump, rAutoSpeed := "Pumps".Pump_1.rAutoSpeedPump, bПускатели := 1, bDriveRunning := "DI".DI_15.f_DI_out, bDriveFault :=, rMinSpeed :=, rMaxSpeed :=, bResetFault := "Pumps".Pump_1.bresAlarm, bRunCmd => "Преобразователь частоты 1 пуск", iSpeedOut => "AO_0.0_Преобразователь частоты 1", "rSpeedHMI(0-100)" => "Pumps".Pump_1.rHMI_Speed, bPumpRunning => "Pumps".Pump_1.bHMI_PumpRun, bPumpFault => "Alarms".Pump_Alarm[1].ALARM, iStatus => "Pumps".Pump_1.iStatusPump)
   END_RUNG
   RUNG wire#powerrail
      I_Contact( "Pumps".Pump_1.bManualStart )
   END_RUNG wire#w1
   RUNG wire#powerrail
      I_Contact( "Pumps".Pump_1.bAutoStartPump )
   END_RUNG wire#w2
   RUNG wire#powerrail
      I_Contact( "Alarms".Avtomat_Off[1].ALARM )
   END_RUNG wire#w3
   // the same network as SCL:
   "Pump_1_DB"(bManualMode := "Pumps".Pump_1.bManualMode,   // "Pump"
               bManualStart := "Pumps".Pump_1.bManualStart,
               bManualStop := NOT "Pumps".Pump_1.bManualStart,
               rManualSpeed := "Pumps".Pump_1.rManualSpeed,
               bDryRunn := "LS"."LS-1",
               bAutoSTop := NOT "Pumps".Pump_1.bAutoStartPump,
               bAutoStartPerm := "Pumps".Pump_1.bAutoStartPump,
               rAutoSpeed := "Pumps".Pump_1.rAutoSpeedPump,
               bАвтоматы := NOT "Alarms".Avtomat_Off[1].ALARM,
               bПускатели := 1,
               bDriveRunning := "DI".DI_15.f_DI_out,
               bResetFault := "Pumps".Pump_1.bresAlarm,
               bRunCmd => "Преобразователь частоты 1 пуск",
               iSpeedOut => "AO_0.0_Преобразователь частоты 1",
               "rSpeedHMI(0-100)" => "Pumps".Pump_1.rHMI_Speed,
               bPumpRunning => "Pumps".Pump_1.bHMI_PumpRun,
               bPumpFault => "Alarms".Pump_Alarm[1].ALARM,
               iStatus => "Pumps".Pump_1.iStatusPump);
END_REGION

REGION Network 2 (SCL): Контроль сухого хода
   // Контроль по датчику давления если ниже уставки - то сухой ход
   //Detect DrySensor Pump-1
   "IEC_Timer_DetectDry_1".TON(IN := "DB2_HMI_SET".rDetectDry_PressTank1_SP > "AI_DB".PT_01.rAI_Value,
                               PT := "DB2_HMI_SET".diTimeDetectDrt * 1000);
   //Res DrySensot Pump-1
   "IEC_Timer_ResDrySens".TON(IN := "DB2_HMI_SET".rDetectDry_PressTank1_SP < "AI_DB".PT_01.rAI_Value,
                              PT := "DB2_HMI_SET".diTimeDetectDrt * 1000);

   //Фиксация и сброс детектора сухого хода
   IF "IEC_Timer_DetectDry_1".Q THEN
       "bDryContrlPump_1" := TRUE;
   ELSIF "IEC_Timer_ResDrySens".Q THEN
       "bDryContrlPump_1" := FALSE;
   END_IF;
END_REGION

REGION Network 3: Насос 2
   // Привязать датчик давления с уставкой для контроля сухого хода
   RUNG wire#powerrail
      "Pump_2_DB"(bManualStop := wire#w1, bAutoSTop := wire#w2, bAutoStartPerm := wire#w3, bАвтоматы := wire#w4, bManualMode := "Pumps".Pump_2.bManualMode, bManualStart := "Pumps".Pump_2.bManualStart, rManualSpeed := "Pumps".Pump_2.rManualSpeed, bDryRunn := "LS"."LS-2", rAutoSpeed := "Pumps".Pump_2.rAutoSpeedPump, bПускатели := 1, bDriveRunning := "DI".DI_17.f_DI_out, bDriveFault :=, rMinSpeed :=, rMaxSpeed :=, bResetFault := "Pumps".Pump_2.bresAlarm, bRunCmd => "Преобразователь частоты 2 пуск", iSpeedOut => "AO_0.1_Преобразователь частоты 2", "rSpeedHMI(0-100)" => "Pumps".Pump_2.rHMI_Speed, bPumpRunning => "Pumps".Pump_2.bHMI_PumpRun, bPumpFault => "Alarms".Pump_Alarm[2].ALARM, iStatus => "Pumps".Pump_2.iStatusPump)
   END_RUNG
   RUNG wire#powerrail
      I_Contact( "Pumps".Pump_2.bManualStart )
   END_RUNG wire#w1
   RUNG wire#powerrail
      I_Contact( "bStartWork_Main" )
   END_RUNG wire#w2
   RUNG wire#powerrail
      Contact( "bStartWork_Main" )
   END_RUNG wire#w3
   RUNG wire#powerrail
      I_Contact( "Alarms".Avtomat_Off[2].ALARM )
   END_RUNG wire#w4
   // the same network as SCL:
   "Pump_2_DB"(bManualMode := "Pumps".Pump_2.bManualMode,   // "Pump"
               bManualStart := "Pumps".Pump_2.bManualStart,
               bManualStop := NOT "Pumps".Pump_2.bManualStart,
               rManualSpeed := "Pumps".Pump_2.rManualSpeed,
               bDryRunn := "LS"."LS-2",
               bAutoSTop := NOT "bStartWork_Main",
               bAutoStartPerm := "bStartWork_Main",
               rAutoSpeed := "Pumps".Pump_2.rAutoSpeedPump,
               bАвтоматы := NOT "Alarms".Avtomat_Off[2].ALARM,
               bПускатели := 1,
               bDriveRunning := "DI".DI_17.f_DI_out,
               bResetFault := "Pumps".Pump_2.bresAlarm,
               bRunCmd => "Преобразователь частоты 2 пуск",
               iSpeedOut => "AO_0.1_Преобразователь частоты 2",
               "rSpeedHMI(0-100)" => "Pumps".Pump_2.rHMI_Speed,
               bPumpRunning => "Pumps".Pump_2.bHMI_PumpRun,
               bPumpFault => "Alarms".Pump_Alarm[2].ALARM,
               iStatus => "Pumps".Pump_2.iStatusPump);
END_REGION
END_FUNCTION

FUNCTION "Analogs_IN_All" : Void   // FC6, LAD
TITLE = Датчики AI
{ S7_Optimized_Access := 'FALSE' }
VERSION : 0.1
BEGIN

REGION Network 1: Датчик температуры - 1
   // TT-01
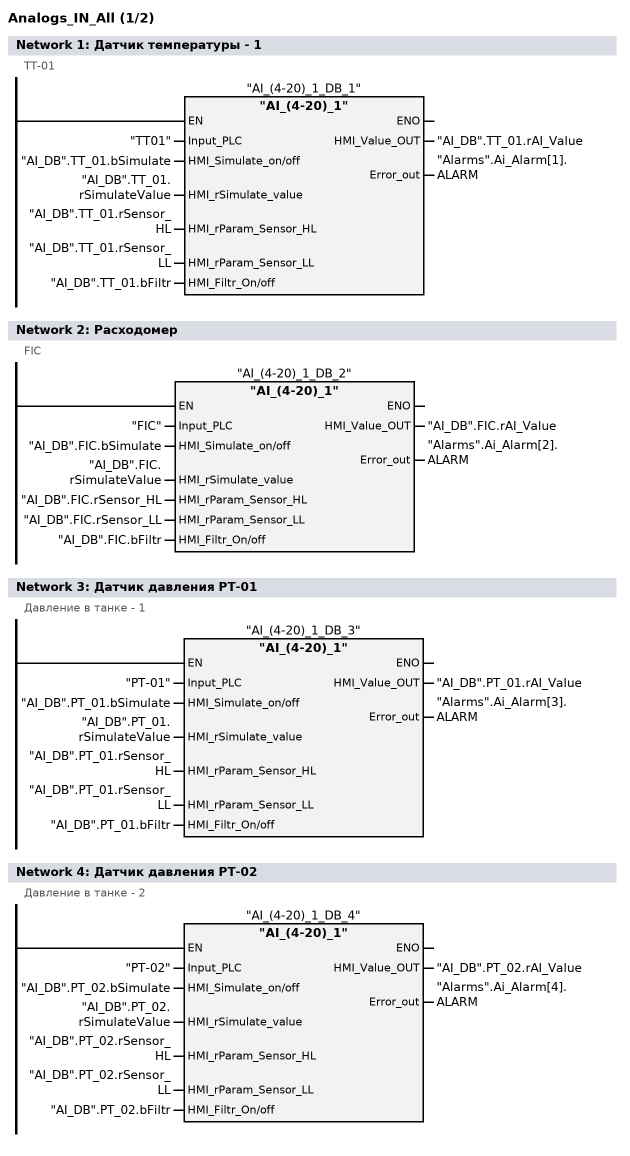
   RUNG wire#powerrail
      "AI_(4-20)_1_DB_1"(Input_PLC := "ТТ01", "HMI_Simulate_on/off" := "AI_DB".TT_01.bSimulate, HMI_rSimulate_value := "AI_DB".TT_01.rSimulateValue, HMI_rParam_Sensor_HL := "AI_DB".TT_01.rSensor_HL, HMI_rParam_Sensor_LL := "AI_DB".TT_01.rSensor_LL, "HMI_Filtr_On/off" := "AI_DB".TT_01.bFiltr, HMI_Value_OUT => "AI_DB".TT_01.rAI_Value, Error_out => "Alarms".Ai_Alarm[1].ALARM)
   END_RUNG
   // the same network as SCL:
   "AI_(4-20)_1_DB_1"(Input_PLC := "ТТ01",   // "AI_(4-20)_1"
                      "HMI_Simulate_on/off" := "AI_DB".TT_01.bSimulate,
                      HMI_rSimulate_value := "AI_DB".TT_01.rSimulateValue,
                      HMI_rParam_Sensor_HL := "AI_DB".TT_01.rSensor_HL,
                      HMI_rParam_Sensor_LL := "AI_DB".TT_01.rSensor_LL,
                      "HMI_Filtr_On/off" := "AI_DB".TT_01.bFiltr,
                      HMI_Value_OUT => "AI_DB".TT_01.rAI_Value,
                      Error_out => "Alarms".Ai_Alarm[1].ALARM);
END_REGION

REGION Network 2: Расходомер
   // FIC
   RUNG wire#powerrail
      "AI_(4-20)_1_DB_2"(Input_PLC := "FIC", "HMI_Simulate_on/off" := "AI_DB".FIC.bSimulate, HMI_rSimulate_value := "AI_DB".FIC.rSimulateValue, HMI_rParam_Sensor_HL := "AI_DB".FIC.rSensor_HL, HMI_rParam_Sensor_LL := "AI_DB".FIC.rSensor_LL, "HMI_Filtr_On/off" := "AI_DB".FIC.bFiltr, HMI_Value_OUT => "AI_DB".FIC.rAI_Value, Error_out => "Alarms".Ai_Alarm[2].ALARM)
   END_RUNG
   // the same network as SCL:
   "AI_(4-20)_1_DB_2"(Input_PLC := "FIC",   // "AI_(4-20)_1"
                      "HMI_Simulate_on/off" := "AI_DB".FIC.bSimulate,
                      HMI_rSimulate_value := "AI_DB".FIC.rSimulateValue,
                      HMI_rParam_Sensor_HL := "AI_DB".FIC.rSensor_HL,
                      HMI_rParam_Sensor_LL := "AI_DB".FIC.rSensor_LL,
                      "HMI_Filtr_On/off" := "AI_DB".FIC.bFiltr,
                      HMI_Value_OUT => "AI_DB".FIC.rAI_Value,
                      Error_out => "Alarms".Ai_Alarm[2].ALARM);
END_REGION

REGION Network 3: Датчик давления РТ-01
   // Давление в танке - 1
   RUNG wire#powerrail
      "AI_(4-20)_1_DB_3"(Input_PLC := "PT-01", "HMI_Simulate_on/off" := "AI_DB".PT_01.bSimulate, HMI_rSimulate_value := "AI_DB".PT_01.rSimulateValue, HMI_rParam_Sensor_HL := "AI_DB".PT_01.rSensor_HL, HMI_rParam_Sensor_LL := "AI_DB".PT_01.rSensor_LL, "HMI_Filtr_On/off" := "AI_DB".PT_01.bFiltr, HMI_Value_OUT => "AI_DB".PT_01.rAI_Value, Error_out => "Alarms".Ai_Alarm[3].ALARM)
   END_RUNG
   // the same network as SCL:
   "AI_(4-20)_1_DB_3"(Input_PLC := "PT-01",   // "AI_(4-20)_1"
                      "HMI_Simulate_on/off" := "AI_DB".PT_01.bSimulate,
                      HMI_rSimulate_value := "AI_DB".PT_01.rSimulateValue,
                      HMI_rParam_Sensor_HL := "AI_DB".PT_01.rSensor_HL,
                      HMI_rParam_Sensor_LL := "AI_DB".PT_01.rSensor_LL,
                      "HMI_Filtr_On/off" := "AI_DB".PT_01.bFiltr,
                      HMI_Value_OUT => "AI_DB".PT_01.rAI_Value,
                      Error_out => "Alarms".Ai_Alarm[3].ALARM);
END_REGION

REGION Network 4: Датчик давления РТ-02
   // Давление в танке - 2
   RUNG wire#powerrail
      "AI_(4-20)_1_DB_4"(Input_PLC := "PT-02", "HMI_Simulate_on/off" := "AI_DB".PT_02.bSimulate, HMI_rSimulate_value := "AI_DB".PT_02.rSimulateValue, HMI_rParam_Sensor_HL := "AI_DB".PT_02.rSensor_HL, HMI_rParam_Sensor_LL := "AI_DB".PT_02.rSensor_LL, "HMI_Filtr_On/off" := "AI_DB".PT_02.bFiltr, HMI_Value_OUT => "AI_DB".PT_02.rAI_Value, Error_out => "Alarms".Ai_Alarm[4].ALARM)
   END_RUNG
   // the same network as SCL:
   "AI_(4-20)_1_DB_4"(Input_PLC := "PT-02",   // "AI_(4-20)_1"
                      "HMI_Simulate_on/off" := "AI_DB".PT_02.bSimulate,
                      HMI_rSimulate_value := "AI_DB".PT_02.rSimulateValue,
                      HMI_rParam_Sensor_HL := "AI_DB".PT_02.rSensor_HL,
                      HMI_rParam_Sensor_LL := "AI_DB".PT_02.rSensor_LL,
                      "HMI_Filtr_On/off" := "AI_DB".PT_02.bFiltr,
                      HMI_Value_OUT => "AI_DB".PT_02.rAI_Value,
                      Error_out => "Alarms".Ai_Alarm[4].ALARM);
END_REGION

REGION Network 5: Датчик давления РТ-03
   // Датчик давления на выходе из такнка-2
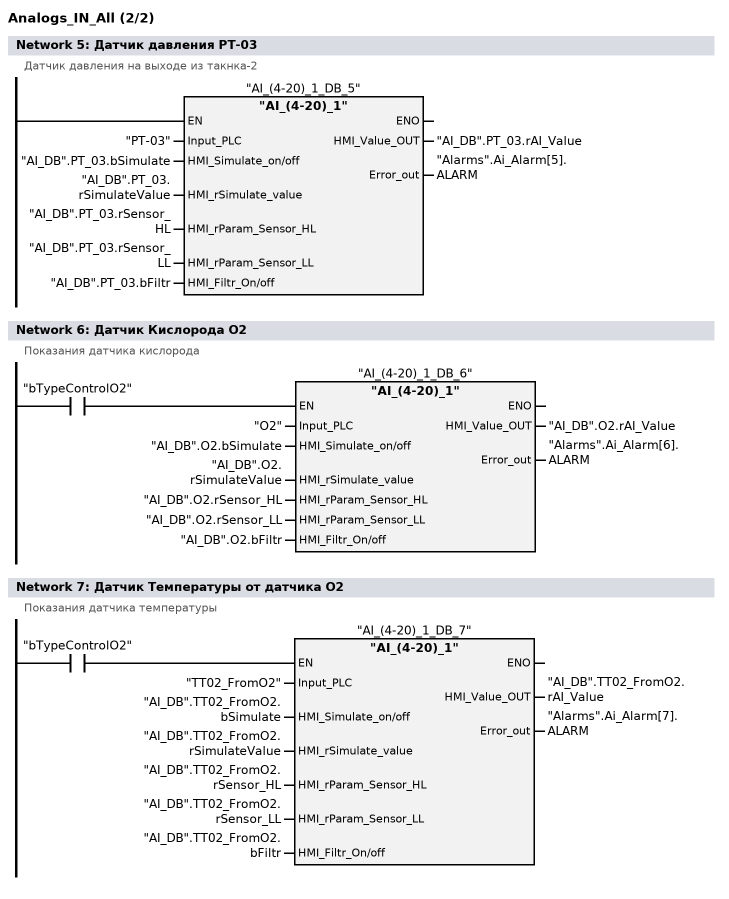
   RUNG wire#powerrail
      "AI_(4-20)_1_DB_5"(Input_PLC := "PT-03", "HMI_Simulate_on/off" := "AI_DB".PT_03.bSimulate, HMI_rSimulate_value := "AI_DB".PT_03.rSimulateValue, HMI_rParam_Sensor_HL := "AI_DB".PT_03.rSensor_HL, HMI_rParam_Sensor_LL := "AI_DB".PT_03.rSensor_LL, "HMI_Filtr_On/off" := "AI_DB".PT_03.bFiltr, HMI_Value_OUT => "AI_DB".PT_03.rAI_Value, Error_out => "Alarms".Ai_Alarm[5].ALARM)
   END_RUNG
   // the same network as SCL:
   "AI_(4-20)_1_DB_5"(Input_PLC := "PT-03",   // "AI_(4-20)_1"
                      "HMI_Simulate_on/off" := "AI_DB".PT_03.bSimulate,
                      HMI_rSimulate_value := "AI_DB".PT_03.rSimulateValue,
                      HMI_rParam_Sensor_HL := "AI_DB".PT_03.rSensor_HL,
                      HMI_rParam_Sensor_LL := "AI_DB".PT_03.rSensor_LL,
                      "HMI_Filtr_On/off" := "AI_DB".PT_03.bFiltr,
                      HMI_Value_OUT => "AI_DB".PT_03.rAI_Value,
                      Error_out => "Alarms".Ai_Alarm[5].ALARM);
END_REGION

REGION Network 6: Датчик Кислорода О2
   // Показания датчика кислорода
   RUNG wire#powerrail
      Contact( "bTypeControlO2" )
      "AI_(4-20)_1_DB_6"(Input_PLC := "O2", "HMI_Simulate_on/off" := "AI_DB".O2.bSimulate, HMI_rSimulate_value := "AI_DB".O2.rSimulateValue, HMI_rParam_Sensor_HL := "AI_DB".O2.rSensor_HL, HMI_rParam_Sensor_LL := "AI_DB".O2.rSensor_LL, "HMI_Filtr_On/off" := "AI_DB".O2.bFiltr, HMI_Value_OUT => "AI_DB".O2.rAI_Value, Error_out => "Alarms".Ai_Alarm[6].ALARM)
   END_RUNG
   // the same network as SCL:
   IF "bTypeControlO2" THEN
       "AI_(4-20)_1_DB_6"(Input_PLC := "O2",   // "AI_(4-20)_1"
                          "HMI_Simulate_on/off" := "AI_DB".O2.bSimulate,
                          HMI_rSimulate_value := "AI_DB".O2.rSimulateValue,
                          HMI_rParam_Sensor_HL := "AI_DB".O2.rSensor_HL,
                          HMI_rParam_Sensor_LL := "AI_DB".O2.rSensor_LL,
                          "HMI_Filtr_On/off" := "AI_DB".O2.bFiltr,
                          HMI_Value_OUT => "AI_DB".O2.rAI_Value,
                          Error_out => "Alarms".Ai_Alarm[6].ALARM);
   END_IF;
END_REGION

REGION Network 7: Датчик Температуры от датчика О2
   // Показания датчика температуры
   RUNG wire#powerrail
      Contact( "bTypeControlO2" )
      "AI_(4-20)_1_DB_7"(Input_PLC := "ТТ02_FromO2", "HMI_Simulate_on/off" := "AI_DB".ТТ02_FromO2.bSimulate, HMI_rSimulate_value := "AI_DB".ТТ02_FromO2.rSimulateValue, HMI_rParam_Sensor_HL := "AI_DB".ТТ02_FromO2.rSensor_HL, HMI_rParam_Sensor_LL := "AI_DB".ТТ02_FromO2.rSensor_LL, "HMI_Filtr_On/off" := "AI_DB".ТТ02_FromO2.bFiltr, HMI_Value_OUT => "AI_DB".ТТ02_FromO2.rAI_Value, Error_out => "Alarms".Ai_Alarm[7].ALARM)
   END_RUNG
   // the same network as SCL:
   IF "bTypeControlO2" THEN
       "AI_(4-20)_1_DB_7"(Input_PLC := "ТТ02_FromO2",   // "AI_(4-20)_1"
                          "HMI_Simulate_on/off" := "AI_DB".ТТ02_FromO2.bSimulate,
                          HMI_rSimulate_value := "AI_DB".ТТ02_FromO2.rSimulateValue,
                          HMI_rParam_Sensor_HL := "AI_DB".ТТ02_FromO2.rSensor_HL,
                          HMI_rParam_Sensor_LL := "AI_DB".ТТ02_FromO2.rSensor_LL,
                          "HMI_Filtr_On/off" := "AI_DB".ТТ02_FromO2.bFiltr,
                          HMI_Value_OUT => "AI_DB".ТТ02_FromO2.rAI_Value,
                          Error_out => "Alarms".Ai_Alarm[7].ALARM);
   END_IF;
END_REGION
END_FUNCTION

FUNCTION "Discret_Inputs_All" : Void   // FC8, LAD
TITLE = Для сбора всех DI в одном месте
{ S7_Optimized_Access := 'FALSE' }
VERSION : 0.1
   VAR CONSTANT
      Cons_TimeDelay : DInt := 100;
   END_VAR
BEGIN

REGION Network 1: E-Stop1
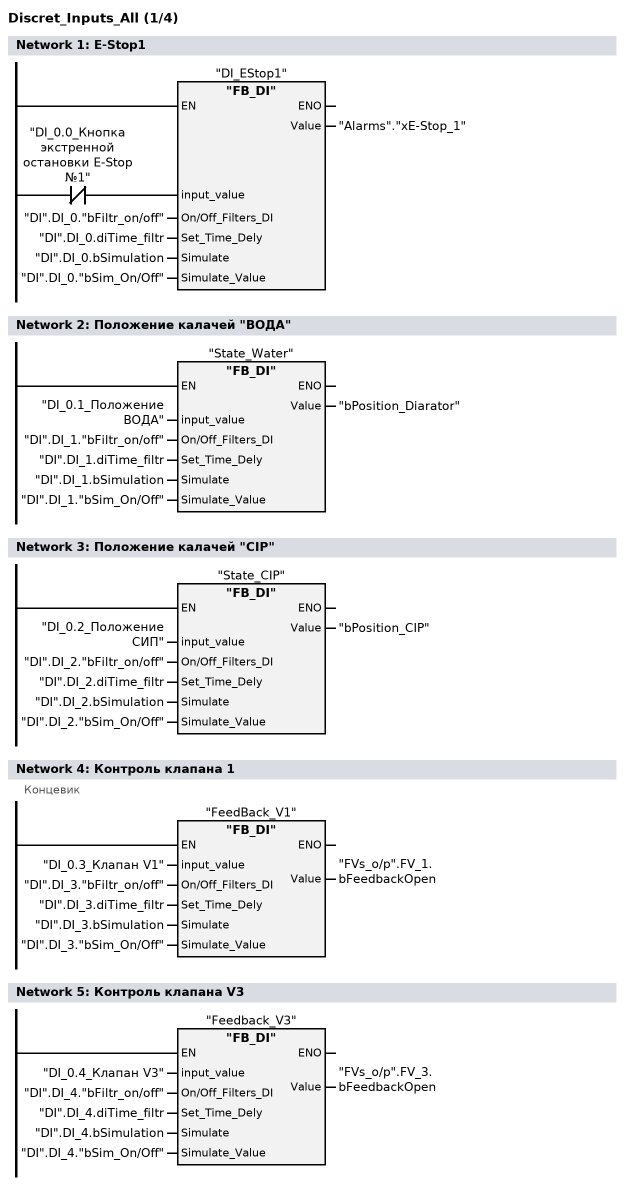
   RUNG wire#powerrail
      "DI_EStop1"(input_value := wire#w1, "On/Off_Filters_DI" := "DI".DI_0."bFiltr_on/off", Set_Time_Dely := "DI".DI_0.diTime_filtr, Simulate := "DI".DI_0.bSimulation, Simulate_Value := "DI".DI_0."bSim_On/Off", Value => "Alarms"."xE-Stop_1")
   END_RUNG
   RUNG wire#powerrail
      I_Contact( "DI_0.0_Кнопка экстренной остановки E-Stop №1" )
   END_RUNG wire#w1
   // the same network as SCL:
   "DI_EStop1"(input_value := NOT "DI_0.0_Кнопка экстренной остановки E-Stop №1",   // "FB_DI"
               "On/Off_Filters_DI" := "DI".DI_0."bFiltr_on/off",
               Set_Time_Dely := "DI".DI_0.diTime_filtr,
               Simulate := "DI".DI_0.bSimulation,
               Simulate_Value := "DI".DI_0."bSim_On/Off",
               Value => "Alarms"."xE-Stop_1");
END_REGION

REGION Network 2: Положение калачей "ВОДА"
   RUNG wire#powerrail
      "State_Water"(input_value := "DI_0.1_Положение ВОДА", "On/Off_Filters_DI" := "DI".DI_1."bFiltr_on/off", Set_Time_Dely := "DI".DI_1.diTime_filtr, Simulate := "DI".DI_1.bSimulation, Simulate_Value := "DI".DI_1."bSim_On/Off", Value => "bPosition_Diarator")
   END_RUNG
   // the same network as SCL:
   "State_Water"(input_value := "DI_0.1_Положение ВОДА",   // "FB_DI"
                 "On/Off_Filters_DI" := "DI".DI_1."bFiltr_on/off",
                 Set_Time_Dely := "DI".DI_1.diTime_filtr,
                 Simulate := "DI".DI_1.bSimulation,
                 Simulate_Value := "DI".DI_1."bSim_On/Off",
                 Value => "bPosition_Diarator");
END_REGION

REGION Network 3: Положение калачей "CIP"
   RUNG wire#powerrail
      "State_CIP"(input_value := "DI_0.2_Положение СИП", "On/Off_Filters_DI" := "DI".DI_2."bFiltr_on/off", Set_Time_Dely := "DI".DI_2.diTime_filtr, Simulate := "DI".DI_2.bSimulation, Simulate_Value := "DI".DI_2."bSim_On/Off", Value => "bPosition_CIP")
   END_RUNG
   // the same network as SCL:
   "State_CIP"(input_value := "DI_0.2_Положение СИП",   // "FB_DI"
               "On/Off_Filters_DI" := "DI".DI_2."bFiltr_on/off",
               Set_Time_Dely := "DI".DI_2.diTime_filtr,
               Simulate := "DI".DI_2.bSimulation,
               Simulate_Value := "DI".DI_2."bSim_On/Off",
               Value => "bPosition_CIP");
END_REGION

REGION Network 4: Контроль клапана 1
   // Концевик
   RUNG wire#powerrail
      "FeedBack_V1"(input_value := "DI_0.3_Клапан V1", "On/Off_Filters_DI" := "DI".DI_3."bFiltr_on/off", Set_Time_Dely := "DI".DI_3.diTime_filtr, Simulate := "DI".DI_3.bSimulation, Simulate_Value := "DI".DI_3."bSim_On/Off", Value => "FVs_o/p".FV_1.bFeedbackOpen)
   END_RUNG
   // the same network as SCL:
   "FeedBack_V1"(input_value := "DI_0.3_Клапан V1",   // "FB_DI"
                 "On/Off_Filters_DI" := "DI".DI_3."bFiltr_on/off",
                 Set_Time_Dely := "DI".DI_3.diTime_filtr,
                 Simulate := "DI".DI_3.bSimulation,
                 Simulate_Value := "DI".DI_3."bSim_On/Off",
                 Value => "FVs_o/p".FV_1.bFeedbackOpen);
END_REGION

REGION Network 5: Контроль клапана V3
   RUNG wire#powerrail
      "Feedback_V3"(input_value := "DI_0.4_Клапан V3", "On/Off_Filters_DI" := "DI".DI_4."bFiltr_on/off", Set_Time_Dely := "DI".DI_4.diTime_filtr, Simulate := "DI".DI_4.bSimulation, Simulate_Value := "DI".DI_4."bSim_On/Off", Value => "FVs_o/p".FV_3.bFeedbackOpen)
   END_RUNG
   // the same network as SCL:
   "Feedback_V3"(input_value := "DI_0.4_Клапан V3",   // "FB_DI"
                 "On/Off_Filters_DI" := "DI".DI_4."bFiltr_on/off",
                 Set_Time_Dely := "DI".DI_4.diTime_filtr,
                 Simulate := "DI".DI_4.bSimulation,
                 Simulate_Value := "DI".DI_4."bSim_On/Off",
                 Value => "FVs_o/p".FV_3.bFeedbackOpen);
END_REGION

REGION Network 6: Контроль клапана V4
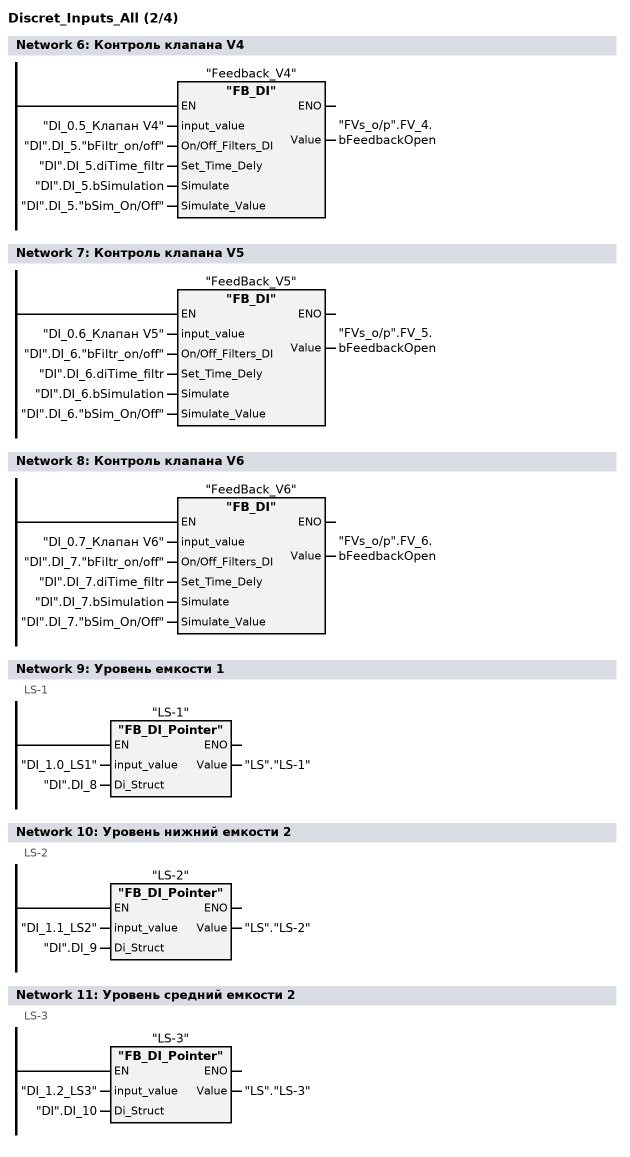
   RUNG wire#powerrail
      "Feedback_V4"(input_value := "DI_0.5_Клапан V4", "On/Off_Filters_DI" := "DI".DI_5."bFiltr_on/off", Set_Time_Dely := "DI".DI_5.diTime_filtr, Simulate := "DI".DI_5.bSimulation, Simulate_Value := "DI".DI_5."bSim_On/Off", Value => "FVs_o/p".FV_4.bFeedbackOpen)
   END_RUNG
   // the same network as SCL:
   "Feedback_V4"(input_value := "DI_0.5_Клапан V4",   // "FB_DI"
                 "On/Off_Filters_DI" := "DI".DI_5."bFiltr_on/off",
                 Set_Time_Dely := "DI".DI_5.diTime_filtr,
                 Simulate := "DI".DI_5.bSimulation,
                 Simulate_Value := "DI".DI_5."bSim_On/Off",
                 Value => "FVs_o/p".FV_4.bFeedbackOpen);
END_REGION

REGION Network 7: Контроль клапана V5
   RUNG wire#powerrail
      "FeedBack_V5"(input_value := "DI_0.6_Клапан V5", "On/Off_Filters_DI" := "DI".DI_6."bFiltr_on/off", Set_Time_Dely := "DI".DI_6.diTime_filtr, Simulate := "DI".DI_6.bSimulation, Simulate_Value := "DI".DI_6."bSim_On/Off", Value => "FVs_o/p".FV_5.bFeedbackOpen)
   END_RUNG
   // the same network as SCL:
   "FeedBack_V5"(input_value := "DI_0.6_Клапан V5",   // "FB_DI"
                 "On/Off_Filters_DI" := "DI".DI_6."bFiltr_on/off",
                 Set_Time_Dely := "DI".DI_6.diTime_filtr,
                 Simulate := "DI".DI_6.bSimulation,
                 Simulate_Value := "DI".DI_6."bSim_On/Off",
                 Value => "FVs_o/p".FV_5.bFeedbackOpen);
END_REGION

REGION Network 8: Контроль клапана V6
   RUNG wire#powerrail
      "FeedBack_V6"(input_value := "DI_0.7_Клапан V6", "On/Off_Filters_DI" := "DI".DI_7."bFiltr_on/off", Set_Time_Dely := "DI".DI_7.diTime_filtr, Simulate := "DI".DI_7.bSimulation, Simulate_Value := "DI".DI_7."bSim_On/Off", Value => "FVs_o/p".FV_6.bFeedbackOpen)
   END_RUNG
   // the same network as SCL:
   "FeedBack_V6"(input_value := "DI_0.7_Клапан V6",   // "FB_DI"
                 "On/Off_Filters_DI" := "DI".DI_7."bFiltr_on/off",
                 Set_Time_Dely := "DI".DI_7.diTime_filtr,
                 Simulate := "DI".DI_7.bSimulation,
                 Simulate_Value := "DI".DI_7."bSim_On/Off",
                 Value => "FVs_o/p".FV_6.bFeedbackOpen);
END_REGION

REGION Network 9: Уровень емкости 1
   // LS-1
   RUNG wire#powerrail
      "LS-1"(input_value := "DI_1.0_LS1", Di_Struct := "DI".DI_8, Value => "LS"."LS-1")
   END_RUNG
   // the same network as SCL:
   "LS-1"(input_value := "DI_1.0_LS1", Di_Struct := "DI".DI_8, Value => "LS"."LS-1");   // "FB_DI_Pointer"
END_REGION

REGION Network 10: Уровень нижний емкости 2
   // LS-2
   RUNG wire#powerrail
      "LS-2"(input_value := "DI_1.1_LS2", Di_Struct := "DI".DI_9, Value => "LS"."LS-2")
   END_RUNG
   // the same network as SCL:
   "LS-2"(input_value := "DI_1.1_LS2", Di_Struct := "DI".DI_9, Value => "LS"."LS-2");   // "FB_DI_Pointer"
END_REGION

REGION Network 11: Уровень средний емкости 2
   // LS-3
   RUNG wire#powerrail
      "LS-3"(input_value := "DI_1.2_LS3", Di_Struct := "DI".DI_10, Value => "LS"."LS-3")
   END_RUNG
   // the same network as SCL:
   "LS-3"(input_value := "DI_1.2_LS3", Di_Struct := "DI".DI_10, Value => "LS"."LS-3");   // "FB_DI_Pointer"
END_REGION

REGION Network 12: Уровень верхний емкости 2
   // LS-4
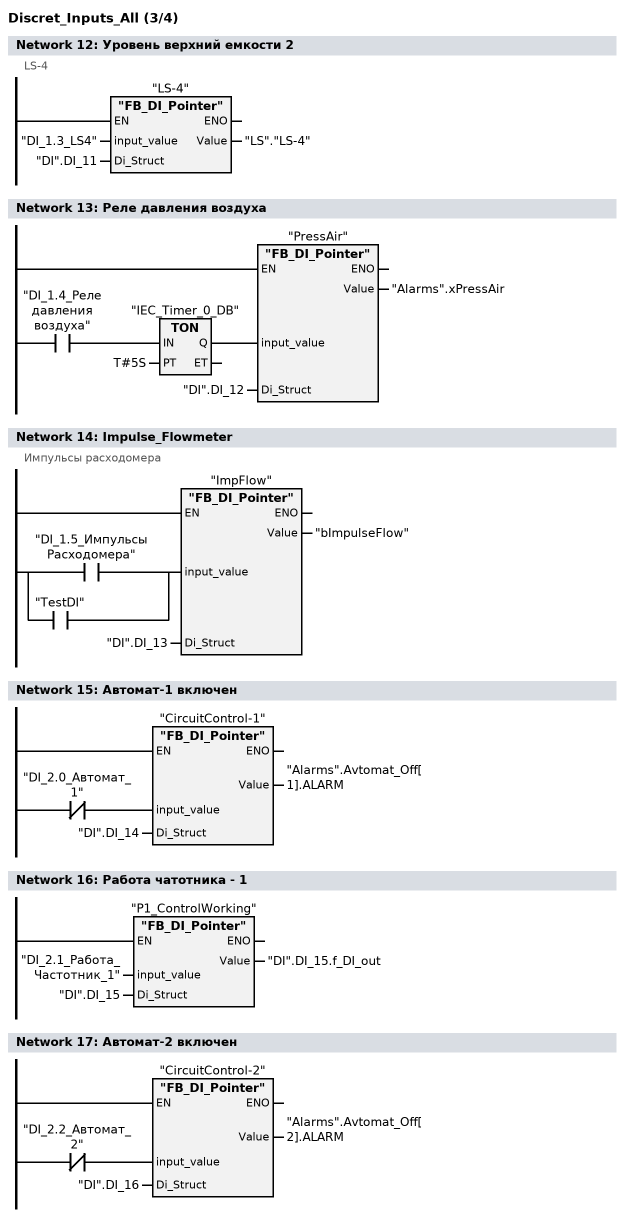
   RUNG wire#powerrail
      "LS-4"(input_value := "DI_1.3_LS4", Di_Struct := "DI".DI_11, Value => "LS"."LS-4")
   END_RUNG
   // the same network as SCL:
   "LS-4"(input_value := "DI_1.3_LS4", Di_Struct := "DI".DI_11, Value => "LS"."LS-4");   // "FB_DI_Pointer"
END_REGION

REGION Network 13: Реле давления воздуха
   "IEC_Timer_0_DB".TON(IN := "DI_1.4_Реле давления воздуха", PT := T#5S);
   "PressAir"(input_value := "IEC_Timer_0_DB".Q, Di_Struct := "DI".DI_12, Value => "Alarms".xPressAir);   // "FB_DI_Pointer"
END_REGION

REGION Network 14: Impulse_Flowmeter
   // Импульсы расходомера
   RUNG wire#powerrail
      "ImpFlow"(input_value := wire#w1, Di_Struct := "DI".DI_13, Value => "bImpulseFlow")
   END_RUNG
   RUNG wire#powerrail
      Contact( "DI_1.5_Импульсы Расходомера" )
   END_RUNG wire#w1
   RUNG wire#powerrail
      Contact( "TestDI" )
   END_RUNG wire#w1
   // the same network as SCL:
   "ImpFlow"(input_value := "DI_1.5_Импульсы Расходомера" OR "TestDI",   // "FB_DI_Pointer"
             Di_Struct := "DI".DI_13,
             Value => "bImpulseFlow");
END_REGION

REGION Network 15: Автомат-1 включен
   RUNG wire#powerrail
      "CircuitControl-1"(input_value := wire#w1, Di_Struct := "DI".DI_14, Value => "Alarms".Avtomat_Off[1].ALARM)
   END_RUNG
   RUNG wire#powerrail
      I_Contact( "DI_2.0_Автомат_1" )
   END_RUNG wire#w1
   // the same network as SCL:
   "CircuitControl-1"(input_value := NOT "DI_2.0_Автомат_1",   // "FB_DI_Pointer"
                      Di_Struct := "DI".DI_14,
                      Value => "Alarms".Avtomat_Off[1].ALARM);
END_REGION

REGION Network 16: Работа чатотника - 1
   RUNG wire#powerrail
      "P1_ControlWorking"(input_value := "DI_2.1_Работа_Частотник_1", Di_Struct := "DI".DI_15, Value => "DI".DI_15.f_DI_out)
   END_RUNG
   // the same network as SCL:
   "P1_ControlWorking"(input_value := "DI_2.1_Работа_Частотник_1",   // "FB_DI_Pointer"
                       Di_Struct := "DI".DI_15,
                       Value => "DI".DI_15.f_DI_out);
END_REGION

REGION Network 17: Автомат-2 включен
   RUNG wire#powerrail
      "CircuitControl-2"(input_value := wire#w1, Di_Struct := "DI".DI_16, Value => "Alarms".Avtomat_Off[2].ALARM)
   END_RUNG
   RUNG wire#powerrail
      I_Contact( "DI_2.2_Автомат_2" )
   END_RUNG wire#w1
   // the same network as SCL:
   "CircuitControl-2"(input_value := NOT "DI_2.2_Автомат_2",   // "FB_DI_Pointer"
                      Di_Struct := "DI".DI_16,
                      Value => "Alarms".Avtomat_Off[2].ALARM);
END_REGION

REGION Network 18: Работа чатотника - 2
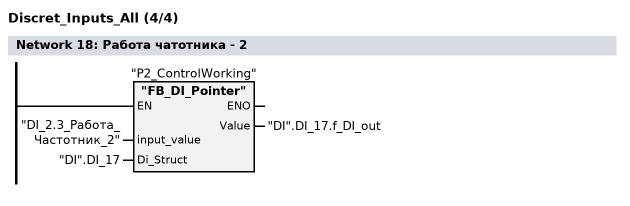
   RUNG wire#powerrail
      "P2_ControlWorking"(input_value := "DI_2.3_Работа_Частотник_2", Di_Struct := "DI".DI_17, Value => "DI".DI_17.f_DI_out)
   END_RUNG
   // the same network as SCL:
   "P2_ControlWorking"(input_value := "DI_2.3_Работа_Частотник_2",   // "FB_DI_Pointer"
                       Di_Struct := "DI".DI_17,
                       Value => "DI".DI_17.f_DI_out);
END_REGION
END_FUNCTION

FUNCTION "Все в Авто" : Void   // FC12, SCL
{ S7_Optimized_Access := 'TRUE' }
VERSION : 0.1
   VAR_TEMP
      fTrig_All_Auto : Bool;   // Фронт нажития кнопки все в авто
   END_VAR
BEGIN

   //Отлавливаем фронт нажатия клавиши все в авто
   "R_trig_All_Auto"(In:="bAllAuto",
                     Q=>#fTrig_All_Auto);

   //Сбрасываем все ручное в автоматический режим
   //
   IF #fTrig_All_Auto THEN

       //симуляция датчиков аналоговых
       "AI_DB".TT_01.bSimulate := FALSE;
       "AI_DB".FIC.bSimulate := FALSE;
       "AI_DB".PT_01.bSimulate := FALSE;
       "AI_DB".PT_02.bSimulate := FALSE;
       "AI_DB".PT_03.bSimulate := FALSE;
       "AI_DB".O2.bSimulate := FALSE;



       //Управление FV
       "FVs_o/p".FV_1.bManualMode := FALSE;
       "FVs_o/p".FV_2.bManualMode := FALSE;
       "FVs_o/p".FV_3.bManualMode := FALSE;
       "FVs_o/p".FV_4.bManualMode := FALSE;
       "FVs_o/p".FV_5.bManualMode := FALSE;
       "FVs_o/p".FV_6.bManualMode := FALSE;
       "FVs_o/p".FV_7.bManualMode := FALSE;
       "FVs_o/p".FV_8.bManualMode := FALSE;
       "FVs_o/p".FV_9.bManualMode := FALSE;
       "FVs_o/p".FV_10.bManualMode := FALSE;


       //Управление Pumps
       "Pumps".Pump_1.bManualMode := FALSE;
       "Pumps".Pump_2.bManualMode := FALSE;


       //Управление клапанами регул %FV
       "FVs_Regul".FV_Regul_1.bHMI_ManualMode := FALSE;


       //DI

       "DI".DI_0.bSimulation := FALSE;
       "DI".DI_1.bSimulation := FALSE;
       "DI".DI_2.bSimulation := FALSE;
       "DI".DI_3.bSimulation := FALSE;
       "DI".DI_4.bSimulation := FALSE;
       "DI".DI_5.bSimulation := FALSE;
       "DI".DI_6.bSimulation := FALSE;
       "DI".DI_7.bSimulation := FALSE;
       "DI".DI_8.bSimulation := FALSE;
       "DI".DI_9.bSimulation := FALSE;
       "DI".DI_10.bSimulation := FALSE;
       "DI".DI_11.bSimulation := FALSE;
       "DI".DI_12.bSimulation := FALSE;
       "DI".DI_13.bSimulation := FALSE;
       "DI".DI_14.bSimulation := FALSE;
       "DI".DI_15.bSimulation := FALSE;
       "DI".DI_16.bSimulation := FALSE;
       "DI".DI_17.bSimulation := FALSE;
       "DI".DI_18.bSimulation := FALSE;
       "DI".DI_19.bSimulation := FALSE;
       "DI".DI_20.bSimulation := FALSE;
       "DI".DI_21.bSimulation := FALSE;
       "DI".DI_22.bSimulation := FALSE;
       "DI".DI_23.bSimulation := FALSE;
       "DI".DI_24.bSimulation := FALSE;
       "DI".DI_25.bSimulation := FALSE;
       "DI".DI_26.bSimulation := FALSE;
       "DI".DI_27.bSimulation := FALSE;
       "DI".DI_28.bSimulation := FALSE;
       "DI".DI_29.bSimulation := FALSE;

   END_IF;
END_FUNCTION

FUNCTION "RestetAlarms" : Void   // FC13, SCL
{ S7_Optimized_Access := 'TRUE' }
VERSION : 0.1
BEGIN
   IF "bResetAlarmCommon" THEN
       //Сброс аварий насосов
       "Pumps".Pump_1.bresAlarm := TRUE;
       "Pumps".Pump_2.bresAlarm := TRUE;




       //Сброс аварий клапана
       "FVs_o/p".FV_1.bResetAlarm := TRUE;
       "FVs_o/p".FV_2.bResetAlarm := TRUE;
       "FVs_o/p".FV_3.bResetAlarm := TRUE;
       "FVs_o/p".FV_4.bResetAlarm := TRUE;
       "FVs_o/p".FV_5.bResetAlarm := TRUE;
       "FVs_o/p".FV_6.bResetAlarm := TRUE;
       "FVs_o/p".FV_7.bResetAlarm := TRUE;

       //Сброс аварий Датчиков
       //

       "Alarms".Ai_Alarm[6].ALARM := FALSE;
       "Alarms".Ai_Alarm[7].ALARM := FALSE;
       "Alarms".xLongWaitWater := false;


   ELSE
       //Сброс аварий насосов
       "Pumps".Pump_1.bresAlarm := False;
       "Pumps".Pump_2.bresAlarm := False;



       //Сброс аварий клапана
       "FVs_o/p".FV_1.bResetAlarm := False;
       "FVs_o/p".FV_2.bResetAlarm := False;
       "FVs_o/p".FV_3.bResetAlarm := False;
       "FVs_o/p".FV_4.bResetAlarm := False;
       "FVs_o/p".FV_5.bResetAlarm := False;
       "FVs_o/p".FV_6.bResetAlarm := False;
       "FVs_o/p".FV_7.bResetAlarm := False;

   END_IF;
END_FUNCTION

ORGANIZATION_BLOCK "Main"   // OB1, LAD, ProgramCycle
TITLE = "Основкая программа"
{ S7_Optimized_Access := 'TRUE' }
VERSION : 0.1
   VAR_TEMP
      Test1 : Bool;
   END_VAR
BEGIN

REGION Network 1: Аварии
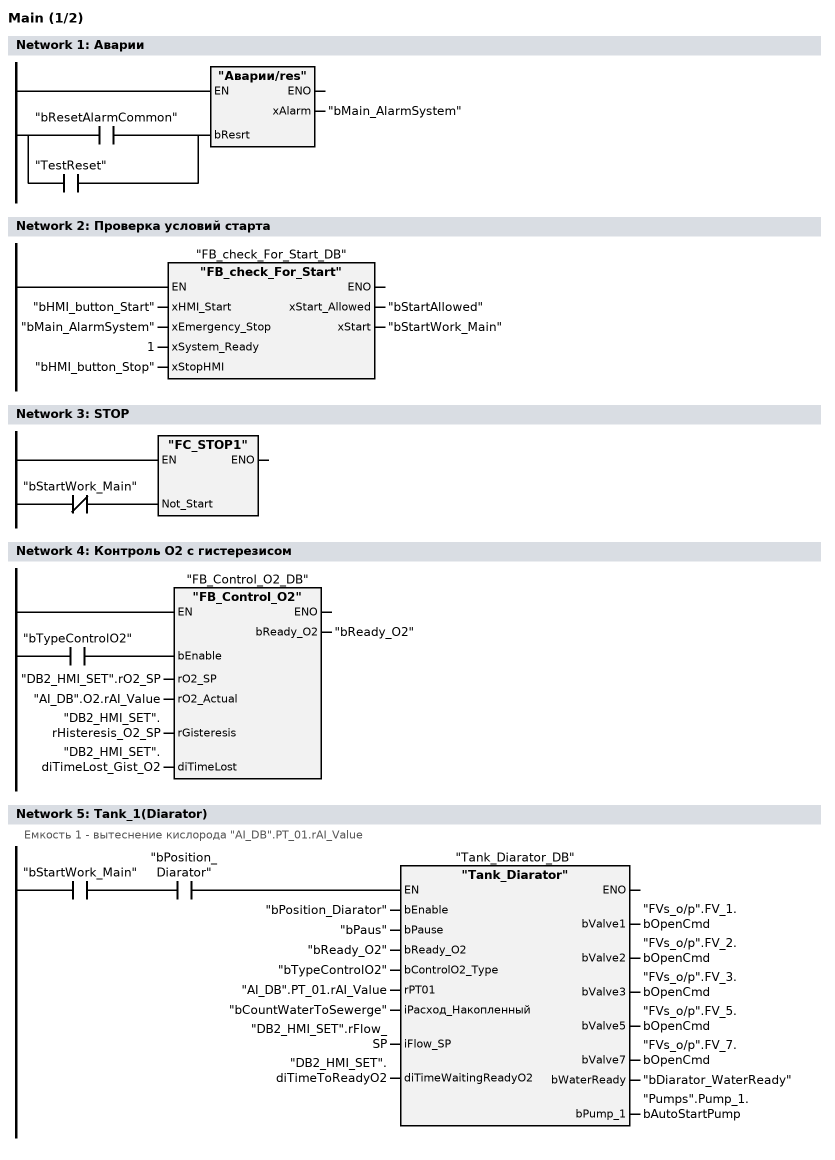
   RUNG wire#powerrail
      "Аварии/res"(bResrt := wire#w1, xAlarm => "bMain_AlarmSystem")
   END_RUNG
   RUNG wire#powerrail
      Contact( "bResetAlarmCommon" )
   END_RUNG wire#w1
   RUNG wire#powerrail
      Contact( "TestReset" )
   END_RUNG wire#w1
   // the same network as SCL:
   "Аварии/res"(bResrt := "bResetAlarmCommon" OR "TestReset", xAlarm => "bMain_AlarmSystem");
END_REGION

REGION Network 2: Проверка условий старта
   RUNG wire#powerrail
      "FB_check_For_Start_DB"(xHMI_Start := "bHMI_button_Start", xEmergency_Stop := "bMain_AlarmSystem", xSystem_Ready := 1, xStopHMI := "bHMI_button_Stop", xStart_Allowed => "bStartAllowed", xStart => "bStartWork_Main")
   END_RUNG
   // the same network as SCL:
   "FB_check_For_Start_DB"(xHMI_Start := "bHMI_button_Start",   // "FB_check_For_Start"
                           xEmergency_Stop := "bMain_AlarmSystem",
                           xSystem_Ready := 1,
                           xStopHMI := "bHMI_button_Stop",
                           xStart_Allowed => "bStartAllowed",
                           xStart => "bStartWork_Main");
END_REGION

REGION Network 3: STOP
   RUNG wire#powerrail
      "FC_STOP1"(Not_Start := wire#w1)
   END_RUNG
   RUNG wire#powerrail
      I_Contact( "bStartWork_Main" )
   END_RUNG wire#w1
   // the same network as SCL:
   "FC_STOP1"(Not_Start := NOT "bStartWork_Main");
END_REGION

REGION Network 4: Контроль О2 с гистерезисом
   RUNG wire#powerrail
      "FB_Control_O2_DB"(bEnable := wire#w1, rO2_SP := "DB2_HMI_SET".rO2_SP, rO2_Actual := "AI_DB".O2.rAI_Value, rGisteresis := "DB2_HMI_SET".rHisteresis_O2_SP, diTimeLost := "DB2_HMI_SET".diTimeLost_Gist_O2, bReady_O2 => "bReady_O2")
   END_RUNG
   RUNG wire#powerrail
      Contact( "bTypeControlO2" )
   END_RUNG wire#w1
   // the same network as SCL:
   "FB_Control_O2_DB"(bEnable := "bTypeControlO2",   // "FB_Control_O2"
                      rO2_SP := "DB2_HMI_SET".rO2_SP,
                      rO2_Actual := "AI_DB".O2.rAI_Value,
                      rGisteresis := "DB2_HMI_SET".rHisteresis_O2_SP,
                      diTimeLost := "DB2_HMI_SET".diTimeLost_Gist_O2,
                      bReady_O2 => "bReady_O2");
END_REGION

REGION Network 5: Tank_1(Diarator)
   // Емкость 1 - вытеснение кислорода "AI_DB".PT_01.rAI_Value
   RUNG wire#powerrail
      Contact( "bStartWork_Main" )
      Contact( "bPosition_Diarator" )
      "Tank_Diarator_DB"(bEnable := "bPosition_Diarator", bPause := "bPaus", bReady_O2 := "bReady_O2", bControlO2_Type := "bTypeControlO2", rPT01 := "AI_DB".PT_01.rAI_Value, iРасход_Накопленный := "bCountWaterToSewerge", iFlow_SP := "DB2_HMI_SET".rFlow_SP, diTimeWaitingReadyO2 := "DB2_HMI_SET".diTimeToReadyO2, bValve1 => "FVs_o/p".FV_1.bOpenCmd, bValve2 => "FVs_o/p".FV_2.bOpenCmd, bValve3 => "FVs_o/p".FV_3.bOpenCmd, bValve5 => "FVs_o/p".FV_5.bOpenCmd, bValve7 => "FVs_o/p".FV_7.bOpenCmd, bWaterReady => "bDiarator_WaterReady", bPump_1 => "Pumps".Pump_1.bAutoStartPump)
   END_RUNG
   // the same network as SCL:
   IF "bStartWork_Main" AND "bPosition_Diarator" THEN
       "Tank_Diarator_DB"(bEnable := "bPosition_Diarator",   // "Tank_Diarator"
                          bPause := "bPaus",
                          bReady_O2 := "bReady_O2",
                          bControlO2_Type := "bTypeControlO2",
                          rPT01 := "AI_DB".PT_01.rAI_Value,
                          iРасход_Накопленный := "bCountWaterToSewerge",
                          iFlow_SP := "DB2_HMI_SET".rFlow_SP,
                          diTimeWaitingReadyO2 := "DB2_HMI_SET".diTimeToReadyO2,
                          bValve1 => "FVs_o/p".FV_1.bOpenCmd,
                          bValve2 => "FVs_o/p".FV_2.bOpenCmd,
                          bValve3 => "FVs_o/p".FV_3.bOpenCmd,
                          bValve5 => "FVs_o/p".FV_5.bOpenCmd,
                          bValve7 => "FVs_o/p".FV_7.bOpenCmd,
                          bWaterReady => "bDiarator_WaterReady",
                          bPump_1 => "Pumps".Pump_1.bAutoStartPump);
   END_IF;
END_REGION

REGION Network 6: Работа Танка-2 (Буфер)
   // Контроль датчиков уровня и таймеры аварии, задержки старта по низкому уровню емкости
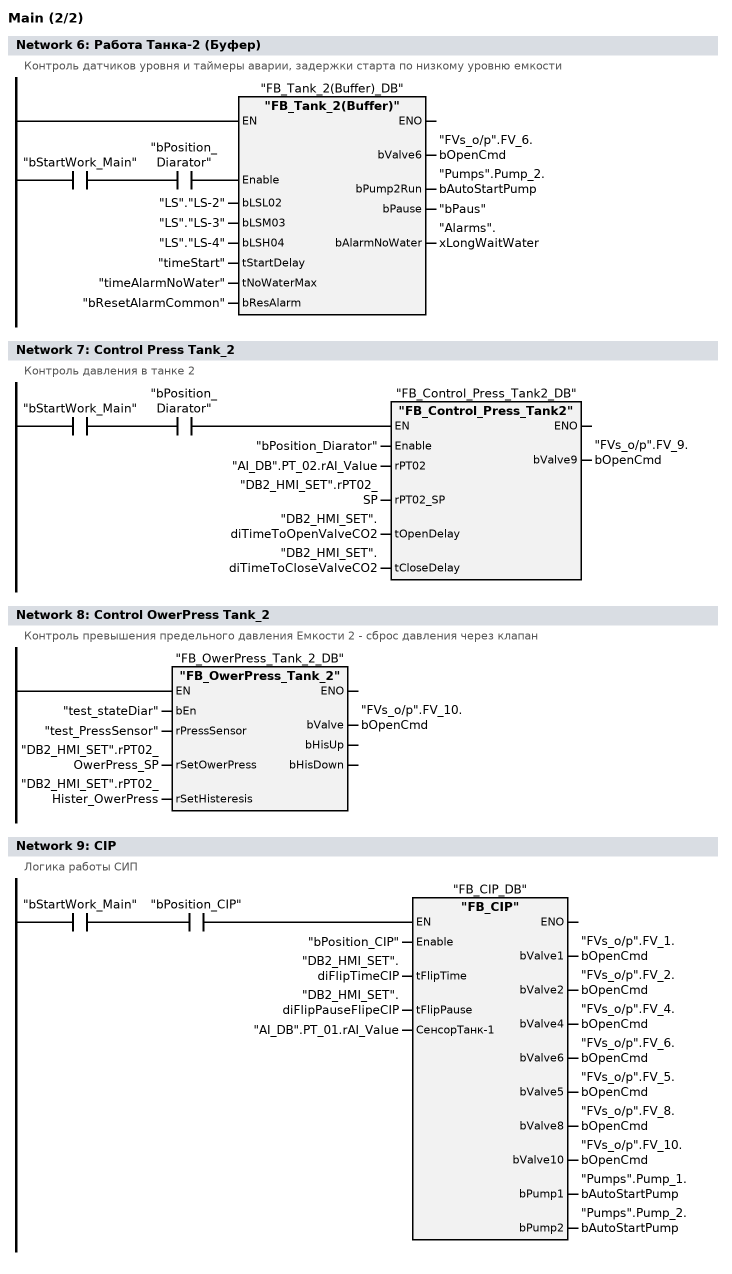
   RUNG wire#powerrail
      "FB_Tank_2(Buffer)_DB"(Enable := wire#w1, bLSL02 := "LS"."LS-2", bLSM03 := "LS"."LS-3", bLSH04 := "LS"."LS-4", tStartDelay := "timeStart", tNoWaterMax := "timeAlarmNoWater", bResAlarm := "bResetAlarmCommon", bValve6 => "FVs_o/p".FV_6.bOpenCmd, bPump2Run => "Pumps".Pump_2.bAutoStartPump, bPause => "bPaus", bAlarmNoWater => "Alarms".xLongWaitWater)
   END_RUNG
   RUNG wire#powerrail
      Contact( "bStartWork_Main" )
      Contact( "bPosition_Diarator" )
   END_RUNG wire#w1
   // the same network as SCL:
   "FB_Tank_2(Buffer)_DB"(Enable := "bStartWork_Main" AND "bPosition_Diarator",   // "FB_Tank_2(Buffer)"
                          bLSL02 := "LS"."LS-2",
                          bLSM03 := "LS"."LS-3",
                          bLSH04 := "LS"."LS-4",
                          tStartDelay := "timeStart",
                          tNoWaterMax := "timeAlarmNoWater",
                          bResAlarm := "bResetAlarmCommon",
                          bValve6 => "FVs_o/p".FV_6.bOpenCmd,
                          bPump2Run => "Pumps".Pump_2.bAutoStartPump,
                          bPause => "bPaus",
                          bAlarmNoWater => "Alarms".xLongWaitWater);
END_REGION

REGION Network 7: Control Press Tank_2
   // Контроль давления в танке 2
   RUNG wire#powerrail
      Contact( "bStartWork_Main" )
      Contact( "bPosition_Diarator" )
      "FB_Control_Press_Tank2_DB"(Enable := "bPosition_Diarator", rPT02 := "AI_DB".PT_02.rAI_Value, rPT02_SP := "DB2_HMI_SET".rPT02_SP, tOpenDelay := "DB2_HMI_SET".diTimeToOpenValveCO2, tCloseDelay := "DB2_HMI_SET".diTimeToCloseValveCO2, bValve9 => "FVs_o/p".FV_9.bOpenCmd)
   END_RUNG
   // the same network as SCL:
   IF "bStartWork_Main" AND "bPosition_Diarator" THEN
       "FB_Control_Press_Tank2_DB"(Enable := "bPosition_Diarator",   // "FB_Control_Press_Tank2"
                               rPT02 := "AI_DB".PT_02.rAI_Value,
                               rPT02_SP := "DB2_HMI_SET".rPT02_SP,
                               tOpenDelay := "DB2_HMI_SET".diTimeToOpenValveCO2,
                               tCloseDelay := "DB2_HMI_SET".diTimeToCloseValveCO2,
                               bValve9 => "FVs_o/p".FV_9.bOpenCmd);
   END_IF;
END_REGION

REGION Network 8: Control OwerPress Tank_2
   // Контроль превышения предельного давления Емкости 2 - сброс давления через клапан
   RUNG wire#powerrail
      "FB_OwerPress_Tank_2_DB"(bEn := "test_stateDiar", rPressSensor := "test_PressSensor", rSetOwerPress := "DB2_HMI_SET".rPT02_OwerPress_SP, rSetHisteresis := "DB2_HMI_SET".rPT02_Hister_OwerPress, bValve => "FVs_o/p".FV_10.bOpenCmd, bHisUp =>, bHisDown =>)
   END_RUNG
   // the same network as SCL:
   "FB_OwerPress_Tank_2_DB"(bEn := "test_stateDiar",   // "FB_OwerPress_Tank_2"
                           rPressSensor := "test_PressSensor",
                           rSetOwerPress := "DB2_HMI_SET".rPT02_OwerPress_SP,
                           rSetHisteresis := "DB2_HMI_SET".rPT02_Hister_OwerPress,
                           bValve => "FVs_o/p".FV_10.bOpenCmd);
END_REGION

REGION Network 9: CIP
   // Логика работы СИП
   RUNG wire#powerrail
      Contact( "bStartWork_Main" )
      Contact( "bPosition_CIP" )
      "FB_CIP_DB"(Enable := "bPosition_CIP", tFlipTime := "DB2_HMI_SET".diFlipTimeCIP, tFlipPause := "DB2_HMI_SET".diFlipPauseFlipeCIP, "СенсорТанк-1" := "AI_DB".PT_01.rAI_Value, bValve1 => "FVs_o/p".FV_1.bOpenCmd, bValve2 => "FVs_o/p".FV_2.bOpenCmd, bValve4 => "FVs_o/p".FV_4.bOpenCmd, bValve6 => "FVs_o/p".FV_6.bOpenCmd, bValve5 => "FVs_o/p".FV_5.bOpenCmd, bValve8 => "FVs_o/p".FV_8.bOpenCmd, bValve10 => "FVs_o/p".FV_10.bOpenCmd, bPump1 => "Pumps".Pump_1.bAutoStartPump, bPump2 => "Pumps".Pump_2.bAutoStartPump)
   END_RUNG
   // the same network as SCL:
   IF "bStartWork_Main" AND "bPosition_CIP" THEN
       "FB_CIP_DB"(Enable := "bPosition_CIP",   // "FB_CIP"
                   tFlipTime := "DB2_HMI_SET".diFlipTimeCIP,
                   tFlipPause := "DB2_HMI_SET".diFlipPauseFlipeCIP,
                   "СенсорТанк-1" := "AI_DB".PT_01.rAI_Value,
                   bValve1 => "FVs_o/p".FV_1.bOpenCmd,
                   bValve2 => "FVs_o/p".FV_2.bOpenCmd,
                   bValve4 => "FVs_o/p".FV_4.bOpenCmd,
                   bValve6 => "FVs_o/p".FV_6.bOpenCmd,
                   bValve5 => "FVs_o/p".FV_5.bOpenCmd,
                   bValve8 => "FVs_o/p".FV_8.bOpenCmd,
                   bValve10 => "FVs_o/p".FV_10.bOpenCmd,
                   bPump1 => "Pumps".Pump_1.bAutoStartPump,
                   bPump2 => "Pumps".Pump_2.bAutoStartPump);
   END_IF;
END_REGION

REGION Network 10 (SCL): Режим работы
   // Для отображения на панели режимов
   IF NOT "bStartWork_Main" THEN
       "iStatusWork" := 0;     //Статус - СТОП
   ELSIF "bStartWork_Main" AND "bPosition_CIP" THEN
       "iStatusWork" := 1;     //Статус - СИП мойка
   ELSIF
       "bStartWork_Main" AND "bPosition_Diarator" AND NOT "bDiarator_WaterReady" THEN
       "iStatusWork" := 2;     //Статус Диарация подготовка воды
   ELSIF
       "bStartWork_Main" AND "bPosition_Diarator" AND "bDiarator_WaterReady" THEN
       "iStatusWork" := 3;     //Статус Диарация - производство
   END_IF;
END_REGION
END_ORGANIZATION_BLOCK

ORGANIZATION_BLOCK "PID"   // OB30, LAD, CyclicInterrupt
{ S7_Optimized_Access := 'TRUE' }
VERSION : 0.1
   VAR_INPUT
      Initial_Call : Bool;   // Initial call of this OB
      Event_Count : Int;   // Events discarded
   END_VAR
   VAR_TEMP   // added for the SCL form of the ladder/FBD networks
      _w1 : Bool;
   END_VAR
BEGIN

REGION Network 1: ПИД - Клапан 2
   // Регулировка по потоку
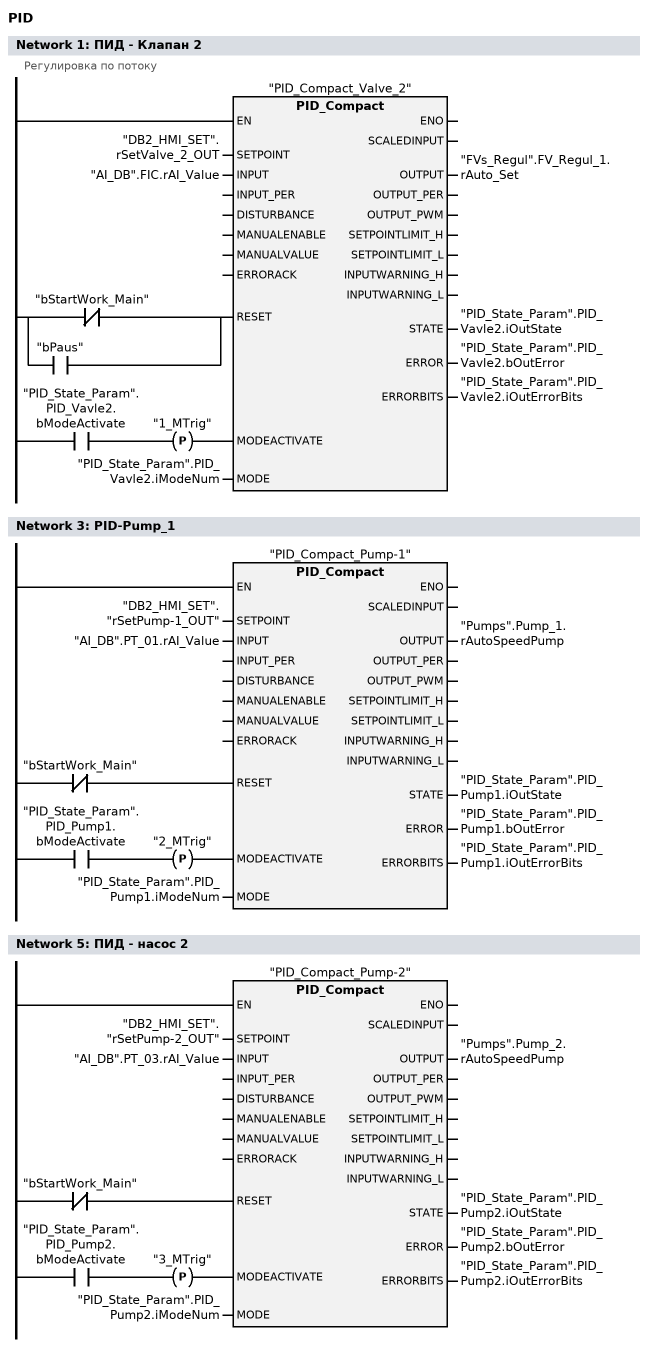
   #_w1 := "PID_State_Param".PID_Vavle2.bModeActivate AND NOT "1_MTrig";   // rising edge
   "1_MTrig" := "PID_State_Param".PID_Vavle2.bModeActivate;
   "PID_Compact_Valve_2"(Setpoint := "DB2_HMI_SET".rSetValve_2_OUT,   // PID_Compact
                         Input := "AI_DB".FIC.rAI_Value,
                         Reset := NOT "bStartWork_Main" OR "bPaus",
                         ModeActivate := #_w1,
                         Mode := "PID_State_Param".PID_Vavle2.iModeNum,
                         Output => "FVs_Regul".FV_Regul_1.rAuto_Set,
                         State => "PID_State_Param".PID_Vavle2.iOutState,
                         Error => "PID_State_Param".PID_Vavle2.bOutError,
                         ErrorBits => "PID_State_Param".PID_Vavle2.iOutErrorBits);
END_REGION

